HMI tags "Default tag table"
   "Any_Alm" : Bool = PLC Any_Alm AT %M6.7, 1 s
   "Reset_All" : Bool = PLC Reset_All AT %M4.1, 1 s
   "settings" : Int AT %DB1.DBW0
   "Any_Hand" : Bool = PLC Any_Hand AT %M5.0, 1 s
   "Logick_hand" : Bool = PLC Logic_DB.Hand AT %DB4.DBX526.7, 1 s
   "Valves_DB_V1_Status" : Int = PLC Valves_DB.V1.Status AT %DB3.DBW10, 1 s
   "Valves_DB_V2_Status" : Int = PLC Valves_DB.V2.Status AT %DB3.DBW134, 1 s
   "AOx_DB_SP_CF_Signal" : Int = PLC AOx_DB.T1_SP.Signal AT %DB8.DBW6, 1 s
   "AOx_DB_SP_CF_SP" : Real = PLC AOx_DB.T1_SP.SP AT %DB8.DBD0, 1 s
   "AOx_DB_SP_CF_CMD_Hand" : Bool = PLC AOx_DB.T1_SP.CMD.Hand AT %DB8.DBX8.0, 1 s
   "AOx_DB_SP_CF_SP_M" : Real = PLC AOx_DB.T1_SP.SP_M AT %DB8.DBD24, 1 s
   "Logic_DB_Start_weight" : Bool = PLC Logic_DB.Start_weight AT %DB4.DBX527.1, 1 s
   "Logic_DB_Alarm" : Word = PLC Logic_DB.Alarm AT %DB4.DBW528, 1 s
   "Motors_DB_T0_Alarm" : Word = PLC Motors_DB.T0.Alarm AT %DB2.DBW34, 1 s
   "Motors_DB_T1_Alarm" : Word = PLC Motors_DB.T1.Alarm AT %DB2.DBW78, 1 s
   "Motors_DB_T2_Alarm" : Word = PLC Motors_DB.T2.Alarm AT %DB2.DBW122, 1 s
   "Motors_DB_T3_Alarm" : Word = PLC Motors_DB.T3.Alarm AT %DB2.DBW166, 1 s
   "Motors_DB_T4_Alarm" : Word = PLC Motors_DB.T4.Alarm AT %DB2.DBW210, 1 s
   "Valves_DB_V1_Alarm" : Word = PLC Valves_DB.V1.Alarm AT %DB3.DBW70, 1 s
   "Valves_DB_V2_Alarm" : Word = PLC Valves_DB.V2.Alarm AT %DB3.DBW194, 1 s
   "Valves_DB_V3_Alarm" : Word = PLC Valves_DB.V3.Alarm AT %DB3.DBW318, 1 s
   "main_screens" : Int AT %DB1.DBW0
   "T4D4_DB_S1_SP" : Real = PLC T4D4_DB.S1.SP AT %DB10.DBD4, 1 s
   "Valves_DB_V1_Delay_On_SP" : Real = PLC Valves_DB.V1.Delay_On.SP AT %DB3.DBD30, 1 s
   "Valves_DB_V1_Delay_On_Now" : Real = PLC Valves_DB.V1.Delay_On.Now AT %DB3.DBD34, 1 s
   "Valves_DB_V1_Delay_Off_SP" : Real = PLC Valves_DB.V1.Delay_Off.SP AT %DB3.DBD48, 1 s
   "Valves_DB_V1_Delay_Off_Now" : Real = PLC Valves_DB.V1.Delay_Off.Now AT %DB3.DBD52, 1 s
   "Vis_reset_stat" : Bool AT %DB1.DBX0.0
   "T2D2_DB_Ready_T3D3" : Bool = PLC T2D2_DB.Ready_T3D3 AT %DB12.DBX0.1, 1 s
   "T3V3W3_DB_Skip_box" : Bool = PLC T3V3W3_DB.Skip_box AT %DB11.DBX8.6, 1 s
   "T3V3W3_DB_SetPoints_SP" : Real = PLC T3V3W3_DB.SetPoints.SP AT %DB11.DBD64, 1 s
   "T3V3W3_DB_LocalVar_SP_loaded" : Real = PLC T3V3W3_DB.LocalVar.SP_loaded AT %DB11.DBD92, 1 s
   "T3V3W3_DB_Reload" : Bool = PLC T3V3W3_DB.Reload AT %DB11.DBX6.4, 1 s
   "T3V3W3_DB_No_box" : Bool = PLC T3V3W3_DB.No_box AT %DB11.DBX8.7, 1 s
   "T3V3W3_DB_Timers_T_s7_SP" : Real = PLC T3V3W3_DB.Timers.T_s7.SP AT %DB11.DBD10, 1 s
   "T3V3W3_DB_Timers_T_s15_SP" : Real = PLC T3V3W3_DB.Timers.T_s15.SP AT %DB11.DBD28, 1 s
   "T3V3W3_DB_SetPoints_SP_ch_s" : Real = PLC T3V3W3_DB.SetPoints.SP_ch_s AT %DB11.DBD72, 1 s
   "T0T1_DB_SP_max" : Real = PLC T0T1_DB.SP_max AT %DB13.DBD8, 1 s
   "T0T1_DB_SP_min" : Real = PLC T0T1_DB.SP_min AT %DB13.DBD4, 1 s
   "T3V3W3_DB_SetPoints_SP_fly" : Real = PLC T3V3W3_DB.SetPoints.SP_fly AT %DB11.DBD68, 1 s
   "T3V3W3_DB_SetPoints_delta_add" : Real = PLC T3V3W3_DB.SetPoints.delta_add AT %DB11.DBD76, 1 s
   "T3V3W3_DB_SetPoints_delata_sub" : Real = PLC T3V3W3_DB.SetPoints.delata_sub AT %DB11.DBD80, 1 s
   "T3V3W3_DB_Reset_weight" : Bool = PLC T3V3W3_DB.Reset_weight AT %DB11.DBX8.4, 1 s
   "T3V3W3_DB_LocalVar_Sp_start" : Real = PLC T3V3W3_DB.LocalVar.Sp_start AT %DB11.DBD104, 1 s
   "Statistic_DB_move_stat_Instance_In_the_beggin" : Bool = PLC Statistic_DB.move_stat_Instance.In_the_beggin AT %DB19.DBX0.0, 1 s
   "Statistic_DB_move_stat_Instance_up" : Bool = PLC Statistic_DB.move_stat_Instance.up AT %DB19.DBX0.2, 1 s
   "T3V3W3_DB_Reset_statistic" : Bool = PLC T3V3W3_DB.Reset_statistic AT %DB11.DBX8.1, 1 s
   "Statistic_DB_move_stat_Instance_down" : Bool = PLC Statistic_DB.move_stat_Instance.down AT %DB19.DBX0.1, 1 s
   "Statistic_DB_move_stat_Instance_box_weight{1}" : Real = PLC Statistic_DB.move_stat_Instance.box_weight[1] AT %DB19.DBD2, 1 s
   "Statistic_DB_move_stat_Instance_box_weight{2}" : Real = PLC Statistic_DB.move_stat_Instance.box_weight[2] AT %DB19.DBD6, 1 s
   "Statistic_DB_move_stat_Instance_box_weight{3}" : Real = PLC Statistic_DB.move_stat_Instance.box_weight[3] AT %DB19.DBD10, 1 s
   "Statistic_DB_move_stat_Instance_box_weight{4}" : Real = PLC Statistic_DB.move_stat_Instance.box_weight[4] AT %DB19.DBD14, 1 s
   "Statistic_DB_move_stat_Instance_box_weight{5}" : Real = PLC Statistic_DB.move_stat_Instance.box_weight[5] AT %DB19.DBD18, 1 s
   "Statistic_DB_move_stat_Instance_box_weight{6}" : Real = PLC Statistic_DB.move_stat_Instance.box_weight[6] AT %DB19.DBD22, 1 s
   "Statistic_DB_move_stat_Instance_box_weight{7}" : Real = PLC Statistic_DB.move_stat_Instance.box_weight[7] AT %DB19.DBD26, 1 s
   "Statistic_DB_move_stat_Instance_box_weight{8}" : Real = PLC Statistic_DB.move_stat_Instance.box_weight[8] AT %DB19.DBD30, 1 s
   "Statistic_DB_move_stat_Instance_box_weight{9}" : Real = PLC Statistic_DB.move_stat_Instance.box_weight[9] AT %DB19.DBD34, 1 s
   "Statistic_DB_move_stat_Instance_box_weight{10}" : Real = PLC Statistic_DB.move_stat_Instance.box_weight[10] AT %DB19.DBD38, 1 s
   "Statistic_DB_move_stat_Instance_box_weight{11}" : Real = PLC Statistic_DB.move_stat_Instance.box_weight[11] AT %DB19.DBD42, 1 s
   "Statistic_DB_move_stat_Instance_box_weight{12}" : Real = PLC Statistic_DB.move_stat_Instance.box_weight[12] AT %DB19.DBD46, 1 s
   "Statistic_DB_move_stat_Instance_box_weight{13}" : Real = PLC Statistic_DB.move_stat_Instance.box_weight[13] AT %DB19.DBD50, 1 s
   "Statistic_DB_move_stat_Instance_box_weight{14}" : Real = PLC Statistic_DB.move_stat_Instance.box_weight[14] AT %DB19.DBD54, 1 s
   "Statistic_DB_move_stat_Instance_box_weight{15}" : Real = PLC Statistic_DB.move_stat_Instance.box_weight[15] AT %DB19.DBD58, 1 s
   "Statistic_DB_move_stat_Instance_box_weight{16}" : Real = PLC Statistic_DB.move_stat_Instance.box_weight[16] AT %DB19.DBD62, 1 s
   "Statistic_DB_move_stat_Instance_box_weight{17}" : Real = PLC Statistic_DB.move_stat_Instance.box_weight[17] AT %DB19.DBD66, 1 s
   "Statistic_DB_move_stat_Instance_box_weight{18}" : Real = PLC Statistic_DB.move_stat_Instance.box_weight[18] AT %DB19.DBD70, 1 s
   "Statistic_DB_move_stat_Instance_box_weight{19}" : Real = PLC Statistic_DB.move_stat_Instance.box_weight[19] AT %DB19.DBD74, 1 s
   "Statistic_DB_move_stat_Instance_box_weight{20}" : Real = PLC Statistic_DB.move_stat_Instance.box_weight[20] AT %DB19.DBD78, 1 s
   "Statistic_DB_move_stat_Instance_box_weight{21}" : Real = PLC Statistic_DB.move_stat_Instance.box_weight[21] AT %DB19.DBD82, 1 s
   "Statistic_DB_move_stat_Instance_box_weight{22}" : Real = PLC Statistic_DB.move_stat_Instance.box_weight[22] AT %DB19.DBD86, 1 s
   "Statistic_DB_move_stat_Instance_box_weight{23}" : Real = PLC Statistic_DB.move_stat_Instance.box_weight[23] AT %DB19.DBD90, 1 s
   "Statistic_DB_move_stat_Instance_box_weight{24}" : Real = PLC Statistic_DB.move_stat_Instance.box_weight[24] AT %DB19.DBD94, 1 s
   "Statistic_DB_move_stat_Instance_box_weight{25}" : Real = PLC Statistic_DB.move_stat_Instance.box_weight[25] AT %DB19.DBD98, 1 s
   "T3V3W3_DB_Statistic_Count" : Int = PLC T3V3W3_DB.Statistic.Count AT %DB11.DBW378, 1 s
   "T3V3W3_DB_Statistic_Mid_weight" : Real = PLC T3V3W3_DB.Statistic.Mid_weight AT %DB11.DBD384, 1 s
   "T3V3W3_DB_Statistic_Weight" : Real = PLC T3V3W3_DB.Statistic.Weight AT %DB11.DBD380, 1 s
   "T3V3W3_DB_Statistic_Count_old" : Int = PLC T3V3W3_DB.Statistic.Count_old AT %DB11.DBW388, 1 s
   "T3V3W3_DB_Statistic_Mid_weight_old" : Real = PLC T3V3W3_DB.Statistic.Mid_weight_old AT %DB11.DBD394, 1 s
   "T3V3W3_DB_Statistic_Weight_old" : Real = PLC T3V3W3_DB.Statistic.Weight_old AT %DB11.DBD390, 1 s
   "T3V3W3_DB_Alarm" : Word = PLC T3V3W3_DB.Alarm AT %DB11.DBW404, 1 s
   "T3V3W3_DB_LocalVar_name_part" : String[254] = PLC T3V3W3_DB.LocalVar.name_part AT %DB11.DBX118.0, 1 s
   "Logic_DB_Clear_mem" : Bool = PLC Logic_DB.Clear_mem AT %DB4.DBX2.0, 1 s
   "T3V3W3_DB_part_names{0}" : String[254] = PLC T3V3W3_DB.part_names[0] AT %DB11.DBX422.0, 1 s
   "T3V3W3_DB_part_names{1}" : String[254] = PLC T3V3W3_DB.part_names[1] AT %DB11.DBX678.0, 1 s
   "T3V3W3_DB_part_names{2}" : String[254] = PLC T3V3W3_DB.part_names[2] AT %DB11.DBX934.0, 1 s
   "T3V3W3_DB_part_names{3}" : String[254] = PLC T3V3W3_DB.part_names[3] AT %DB11.DBX1190.0, 1 s
   "T3V3W3_DB_part_names{4}" : String[254] = PLC T3V3W3_DB.part_names[4] AT %DB11.DBX1446.0, 1 s
   "T3V3W3_DB_part_names{5}" : String[254] = PLC T3V3W3_DB.part_names[5] AT %DB11.DBX1702.0, 1 s
   "T3V3W3_DB_part_names{6}" : String[254] = PLC T3V3W3_DB.part_names[6] AT %DB11.DBX1958.0, 1 s
   "T3V3W3_DB_part_names{7}" : String[254] = PLC T3V3W3_DB.part_names[7] AT %DB11.DBX2214.0, 1 s
   "T3V3W3_DB_part_names{8}" : String[254] = PLC T3V3W3_DB.part_names[8] AT %DB11.DBX2470.0, 1 s
   "T3V3W3_DB_part_names{9}" : String[254] = PLC T3V3W3_DB.part_names[9] AT %DB11.DBX2726.0, 1 s
   "T3V3W3_DB_part_names{10}" : String[254] = PLC T3V3W3_DB.part_names[10] AT %DB11.DBX2982.0, 1 s
   "T3V3W3_DB_part_names{11}" : String[254] = PLC T3V3W3_DB.part_names[11] AT %DB11.DBX3238.0, 1 s
   "T3V3W3_DB_part_names{12}" : String[254] = PLC T3V3W3_DB.part_names[12] AT %DB11.DBX3494.0, 1 s
   "T3V3W3_DB_part_names{13}" : String[254] = PLC T3V3W3_DB.part_names[13] AT %DB11.DBX3750.0, 1 s
   "T3V3W3_DB_part_names{14}" : String[254] = PLC T3V3W3_DB.part_names[14] AT %DB11.DBX4006.0, 1 s
   "T3V3W3_DB_part_names{15}" : String[254] = PLC T3V3W3_DB.part_names[15] AT %DB11.DBX4262.0, 1 s
   "T3V3W3_DB_part_names{16}" : String[254] = PLC T3V3W3_DB.part_names[16] AT %DB11.DBX4518.0, 1 s
   "T3V3W3_DB_part_names{17}" : String[254] = PLC T3V3W3_DB.part_names[17] AT %DB11.DBX4774.0, 1 s
   "T3V3W3_DB_part_names{18}" : String[254] = PLC T3V3W3_DB.part_names[18] AT %DB11.DBX5030.0, 1 s
   "T3V3W3_DB_part_names{19}" : String[254] = PLC T3V3W3_DB.part_names[19] AT %DB11.DBX5286.0, 1 s
   "del_stat_mem_DB_del" : Bool = PLC del_stat_mem_DB.del AT %DB14.DBX0.2, 1 s
   "del_stat_mem_DB_number" : Int = PLC del_stat_mem_DB.number AT %DB14.DBW4, 1 s
   "del_stat_mem_DB_Alarm" : Word = PLC del_stat_mem_DB.Alarm AT %DB14.DBW550, 1 s
   "stat_view" : Int AT %DB1.DBW0
   "T3V3W3_DB_Timers_T_St_Start" : Bool = PLC T3V3W3_DB.Timers.T_St.Start AT %DB11.DBX62.1, 1 s

HMI tags "motors"
   "T0_CMD_Hand" : Bool = PLC Motors_DB.T0.CMD.Hand AT %DB2.DBX6.0, 1 s
   "T0_CMD_Force" : Bool = PLC Motors_DB.T0.CMD.Force AT %DB2.DBX6.3, 1 s
   "T0_Res_h" : DInt = PLC Motors_DB.T0.Res_h AT %DB2.DBD36, 1 s
   "T0_Wait_Off_SP" : Int = PLC Motors_DB.T0.Wait_Off.SP AT %DB2.DBW24, 1 s
   "T0_Wait_Off_Now" : Int = PLC Motors_DB.T0.Wait_Off.Now AT %DB2.DBW26, 1 s
   "T0_Wait_On_SP" : Int = PLC Motors_DB.T0.Wait_On.SP AT %DB2.DBW18, 1 s
   "T0_Wait_On_Now" : Int = PLC Motors_DB.T0.Wait_On.Now AT %DB2.DBW20, 1 s
   "T0_FB_Termo" : Bool = PLC Motors_DB.T0.FB_Termo AT %DB2.DBX0.3, 1 s
   "T0_Use_Termo" : Bool = PLC Motors_DB.T0.Use.Termo AT %DB2.DBX12.4, 1 s
   "T0_Use_Serivce" : Bool = PLC Motors_DB.T0.Use.Serivce AT %DB2.DBX12.3, 1 s
   "T0_Use_KM" : Bool = PLC Motors_DB.T0.Use.KM AT %DB2.DBX12.2, 1 s
   "T0_Use_QF" : Bool = PLC Motors_DB.T0.Use.QF AT %DB2.DBX12.1, 1 s
   "T1_CMD_Hand" : Bool = PLC Motors_DB.T1.CMD.Hand AT %DB2.DBX50.0, 1 s
   "T1_CMD_Force" : Bool = PLC Motors_DB.T1.CMD.Force AT %DB2.DBX50.3, 1 s
   "T1_Res_h" : DInt = PLC Motors_DB.T1.Res_h AT %DB2.DBD80, 1 s
   "T1_Wait_Off_SP" : Int = PLC Motors_DB.T1.Wait_Off.SP AT %DB2.DBW68, 1 s
   "T1_Wait_Off_Now" : Int = PLC Motors_DB.T1.Wait_Off.Now AT %DB2.DBW70, 1 s
   "T1_Wait_On_SP" : Int = PLC Motors_DB.T1.Wait_On.SP AT %DB2.DBW62, 1 s
   "T1_Wait_On_Now" : Int = PLC Motors_DB.T1.Wait_On.Now AT %DB2.DBW64, 1 s
   "T1_FB_Termo" : Bool = PLC Motors_DB.T1.FB_Termo AT %DB2.DBX44.3, 1 s
   "T1_Use_Termo" : Bool = PLC Motors_DB.T1.Use.Termo AT %DB2.DBX56.4, 1 s
   "T1_Use_Serivce" : Bool = PLC Motors_DB.T1.Use.Serivce AT %DB2.DBX56.3, 1 s
   "T1_Use_KM" : Bool = PLC Motors_DB.T1.Use.KM AT %DB2.DBX56.2, 1 s
   "T1_Use_QF" : Bool = PLC Motors_DB.T1.Use.QF AT %DB2.DBX56.1, 1 s
   "T3_CMD_Hand" : Bool = PLC Motors_DB.T3.CMD.Hand AT %DB2.DBX138.0, 1 s
   "T3_CMD_Force" : Bool = PLC Motors_DB.T3.CMD.Force AT %DB2.DBX138.3, 1 s
   "T3_Res_h" : DInt = PLC Motors_DB.T3.Res_h AT %DB2.DBD168, 1 s
   "T3_Wait_Off_SP" : Int = PLC Motors_DB.T3.Wait_Off.SP AT %DB2.DBW156, 1 s
   "T3_Wait_Off_Now" : Int = PLC Motors_DB.T3.Wait_Off.Now AT %DB2.DBW158, 1 s
   "T3_FB_Termo" : Bool = PLC Motors_DB.T3.FB_Termo AT %DB2.DBX132.3, 1 s
   "T3_Use_Termo" : Bool = PLC Motors_DB.T3.Use.Termo AT %DB2.DBX144.4, 1 s
   "T3_Use_Serivce" : Bool = PLC Motors_DB.T3.Use.Serivce AT %DB2.DBX144.3, 1 s
   "T3_Use_KM" : Bool = PLC Motors_DB.T3.Use.KM AT %DB2.DBX144.2, 1 s
   "T3_Use_QF" : Bool = PLC Motors_DB.T3.Use.QF AT %DB2.DBX144.1, 1 s
   "T2_CMD_Hand" : Bool = PLC Motors_DB.T2.CMD.Hand AT %DB2.DBX94.0, 1 s
   "T2_CMD_Force" : Bool = PLC Motors_DB.T2.CMD.Force AT %DB2.DBX94.3, 1 s
   "T2_Res_h" : DInt = PLC Motors_DB.T2.Res_h AT %DB2.DBD124, 1 s
   "T2_Wait_Off_Now" : Int = PLC Motors_DB.T2.Wait_Off.Now AT %DB2.DBW114, 1 s
   "T2_Wait_Off_SP" : Int = PLC Motors_DB.T2.Wait_Off.SP AT %DB2.DBW112, 1 s
   "T2_Wait_On_SP" : Int = PLC Motors_DB.T2.Wait_On.SP AT %DB2.DBW106, 1 s
   "T2_Wait_On_Now" : Int = PLC Motors_DB.T2.Wait_On.Now AT %DB2.DBW108, 1 s
   "T2_FB_Termo" : Bool = PLC Motors_DB.T2.FB_Termo AT %DB2.DBX88.3, 1 s
   "T2_Use_Termo" : Bool = PLC Motors_DB.T2.Use.Termo AT %DB2.DBX100.4, 1 s
   "T2_Use_Serivce" : Bool = PLC Motors_DB.T2.Use.Serivce AT %DB2.DBX100.3, 1 s
   "T2_Use_KM" : Bool = PLC Motors_DB.T2.Use.KM AT %DB2.DBX100.2, 1 s
   "T2_Use_QF" : Bool = PLC Motors_DB.T2.Use.QF AT %DB2.DBX100.1, 1 s
   "T3_Wait_On_SP" : Int = PLC Motors_DB.T3.Wait_On.SP AT %DB2.DBW150, 1 s
   "T3_Wait_On_Now" : Int = PLC Motors_DB.T3.Wait_On.Now AT %DB2.DBW152, 1 s
   "T3_FB_QF" : Bool = PLC Motors_DB.T3.FB_QF AT %DB2.DBX132.0, 1 s
   "T3_FB_KM" : Bool = PLC Motors_DB.T3.FB_KM AT %DB2.DBX132.1, 1 s
   "T3_CMD_Service" : Bool = PLC Motors_DB.T3.CMD.Service AT %DB2.DBX138.6, 1 s
   "T3_CMD_Sim" : Bool = PLC Motors_DB.T3.CMD.Sim AT %DB2.DBX139.2, 1 s
   "T3_Status" : Int = PLC Motors_DB.T3.Status AT %DB2.DBW142, 1 s
   "T3_CMD_Start_M" : Bool = PLC Motors_DB.T3.CMD.Start_M AT %DB2.DBX138.2, 1 s
   "T1_FB_QF" : Bool = PLC Motors_DB.T1.FB_QF AT %DB2.DBX44.0, 1 s
   "T1_FB_KM" : Bool = PLC Motors_DB.T1.FB_KM AT %DB2.DBX44.1, 1 s
   "T1_Status" : Int = PLC Motors_DB.T1.Status AT %DB2.DBW54, 1 s
   "T1_CMD_Sim" : Bool = PLC Motors_DB.T1.CMD.Sim AT %DB2.DBX51.2, 1 s
   "T1_CMD_Start_M" : Bool = PLC Motors_DB.T1.CMD.Start_M AT %DB2.DBX50.2, 1 s
   "T0_FB_QF" : Bool = PLC Motors_DB.T0.FB_QF AT %DB2.DBX0.0, 1 s
   "T0_FB_KM" : Bool = PLC Motors_DB.T0.FB_KM AT %DB2.DBX0.1, 1 s
   "T0_CMD_Sim" : Bool = PLC Motors_DB.T0.CMD.Sim AT %DB2.DBX7.2, 1 s
   "T0_CMD_Start_M" : Bool = PLC Motors_DB.T0.CMD.Start_M AT %DB2.DBX6.2, 1 s
   "T0_Status" : Int = PLC Motors_DB.T0.Status AT %DB2.DBW10, 1 s
   "T2_FB_QF" : Bool = PLC Motors_DB.T2.FB_QF AT %DB2.DBX88.0, 1 s
   "T2_FB_KM" : Bool = PLC Motors_DB.T2.FB_KM AT %DB2.DBX88.1, 1 s
   "T2_CMD_Start_M" : Bool = PLC Motors_DB.T2.CMD.Start_M AT %DB2.DBX94.2, 1 s
   "T2_CMD_Sim" : Bool = PLC Motors_DB.T2.CMD.Sim AT %DB2.DBX95.2, 1 s
   "T2_Status" : Int = PLC Motors_DB.T2.Status AT %DB2.DBW98, 1 s
   "T0_CMD_Service" : Bool = PLC Motors_DB.T0.CMD.Service AT %DB2.DBX6.6, 1 s
   "T1_CMD_Service" : Bool = PLC Motors_DB.T1.CMD.Service AT %DB2.DBX50.6, 1 s
   "T2_CMD_Service" : Bool = PLC Motors_DB.T2.CMD.Service AT %DB2.DBX94.6, 1 s
   "T4_FB_QF" : Bool = PLC Motors_DB.T4.FB_QF AT %DB2.DBX176.0, 1 s
   "T4_FB_KM" : Bool = PLC Motors_DB.T4.FB_KM AT %DB2.DBX176.1, 1 s
   "T4_FB_Service" : Bool = PLC Motors_DB.T4.FB_Service AT %DB2.DBX176.2, 1 s
   "T4_FB_Termo" : Bool = PLC Motors_DB.T4.FB_Termo AT %DB2.DBX176.3, 1 s
   "T4_CMD_Hand" : Bool = PLC Motors_DB.T4.CMD.Hand AT %DB2.DBX182.0, 1 s
   "T4_CMD_Start_A" : Bool = PLC Motors_DB.T4.CMD.Start_A AT %DB2.DBX182.1, 1 s
   "T4_CMD_Start_M" : Bool = PLC Motors_DB.T4.CMD.Start_M AT %DB2.DBX182.2, 1 s
   "T4_CMD_Force" : Bool = PLC Motors_DB.T4.CMD.Force AT %DB2.DBX182.3, 1 s
   "T4_CMD_Local" : Bool = PLC Motors_DB.T4.CMD.Local AT %DB2.DBX182.5, 1 s
   "T4_CMD_Safety" : Bool = PLC Motors_DB.T4.CMD.Safety AT %DB2.DBX182.7, 1 s
   "T4_CMD_Service" : Bool = PLC Motors_DB.T4.CMD.Service AT %DB2.DBX182.6, 1 s
   "T4_CMD_Sim" : Bool = PLC Motors_DB.T4.CMD.Sim AT %DB2.DBX183.2, 1 s
   "T4_Status" : Int = PLC Motors_DB.T4.Status AT %DB2.DBW186, 1 s
   "T4_Use_QF" : Bool = PLC Motors_DB.T4.Use.QF AT %DB2.DBX188.1, 1 s
   "T4_Use_KM" : Bool = PLC Motors_DB.T4.Use.KM AT %DB2.DBX188.2, 1 s
   "T4_Use_Serivce" : Bool = PLC Motors_DB.T4.Use.Serivce AT %DB2.DBX188.3, 1 s
   "T4_Use_Termo" : Bool = PLC Motors_DB.T4.Use.Termo AT %DB2.DBX188.4, 1 s
   "T4_FB_QF(1)" : Bool = PLC Motors_DB.T4.FB.QF AT %DB2.DBX190.1, 1 s
   "T4_FB_KM(1)" : Bool = PLC Motors_DB.T4.FB.KM AT %DB2.DBX190.2, 1 s
   "T4_FB_Serivce" : Bool = PLC Motors_DB.T4.FB.Serivce AT %DB2.DBX190.3, 1 s
   "T4_FB_Termo(1)" : Bool = PLC Motors_DB.T4.FB.Termo AT %DB2.DBX190.4, 1 s
   "T4_Wait_On_SP" : Int = PLC Motors_DB.T4.Wait_On.SP AT %DB2.DBW194, 1 s
   "T4_Wait_On_Now" : Int = PLC Motors_DB.T4.Wait_On.Now AT %DB2.DBW196, 1 s
   "T4_Wait_Off_SP" : Int = PLC Motors_DB.T4.Wait_Off.SP AT %DB2.DBW200, 1 s
   "T4_Wait_Off_Now" : Int = PLC Motors_DB.T4.Wait_Off.Now AT %DB2.DBW202, 1 s
   "T4_Res_h" : DInt = PLC Motors_DB.T4.Res_h AT %DB2.DBD212, 1 s

HMI tags "Valves"
   "V1_Status" : Int = PLC Valves_DB.V1.Status AT %DB3.DBW10, 1 s
   "V1_CMD_Force" : Bool = PLC Valves_DB.V1.CMD.Force AT %DB3.DBX6.3, 1 s
   "V1_Wait_On_SP" : Int = PLC Valves_DB.V1.Wait_On.SP AT %DB3.DBW18, 1 s
   "V1_Wait_On_Now" : Int = PLC Valves_DB.V1.Wait_On.Now AT %DB3.DBW20, 1 s
   "V1_CMD_Start_A" : Bool = PLC Valves_DB.V1.CMD.Start_A AT %DB3.DBX6.1, 1 s
   "V1_CMD_Start_M" : Bool = PLC Valves_DB.V1.CMD.Start_M AT %DB3.DBX6.2, 1 s
   "V1_CMD_Hand" : Bool = PLC Valves_DB.V1.CMD.Hand AT %DB3.DBX6.0, 1 s
   "V1_CMD_Service" : Bool = PLC Valves_DB.V1.CMD.Service AT %DB3.DBX6.6, 1 s
   "V1_CMD_Local" : Bool = PLC Valves_DB.V1.CMD.Local AT %DB3.DBX6.5, 1 s
   "V1_Use_QF" : Bool = PLC Valves_DB.V1.Use.QF AT %DB3.DBX12.1, 1 s
   "V1_Use_Serivce" : Bool = PLC Valves_DB.V1.Use.Serivce AT %DB3.DBX12.4, 1 s
   "V1_Use_Open" : Bool = PLC Valves_DB.V1.Use.Open AT %DB3.DBX12.5, 1 s
   "V1_Use_Close" : Bool = PLC Valves_DB.V1.Use.Close AT %DB3.DBX12.6, 1 s
   "V1_FB_QF" : Bool = PLC Valves_DB.V1.FB_QF AT %DB3.DBX0.0, 1 s
   "V1_FB_Open" : Bool = PLC Valves_DB.V1.FB_Open AT %DB3.DBX0.4, 1 s
   "V1_FB_Close" : Bool = PLC Valves_DB.V1.FB_Close AT %DB3.DBX0.5, 1 s
   "V1_FB_Service" : Bool = PLC Valves_DB.V1.FB_Service AT %DB3.DBX0.3, 1 s
   "V1_CMD_Sim" : Bool = PLC Valves_DB.V1.CMD.Sim AT %DB3.DBX7.2, 1 s
   "V1_Res_h" : DInt = PLC Valves_DB.V1.Res_h AT %DB3.DBD72, 1 s
   "V2_FB_QF" : Bool = PLC Valves_DB.V2.FB_QF AT %DB3.DBX124.0, 1 s
   "V2_FB_Service" : Bool = PLC Valves_DB.V2.FB_Service AT %DB3.DBX124.3, 1 s
   "V2_FB_Open" : Bool = PLC Valves_DB.V2.FB_Open AT %DB3.DBX124.4, 1 s
   "V2_FB_Close" : Bool = PLC Valves_DB.V2.FB_Close AT %DB3.DBX124.5, 1 s
   "V2_CMD_Hand" : Bool = PLC Valves_DB.V2.CMD.Hand AT %DB3.DBX130.0, 1 s
   "V2_CMD_Start_M" : Bool = PLC Valves_DB.V2.CMD.Start_M AT %DB3.DBX130.2, 1 s
   "V2_CMD_Force" : Bool = PLC Valves_DB.V2.CMD.Force AT %DB3.DBX130.3, 1 s
   "V2_CMD_Service" : Bool = PLC Valves_DB.V2.CMD.Service AT %DB3.DBX130.6, 1 s
   "V2_CMD_Sim" : Bool = PLC Valves_DB.V2.CMD.Sim AT %DB3.DBX131.2, 1 s
   "V2_Use_QF" : Bool = PLC Valves_DB.V2.Use.QF AT %DB3.DBX136.1, 1 s
   "V2_Use_Serivce" : Bool = PLC Valves_DB.V2.Use.Serivce AT %DB3.DBX136.4, 1 s
   "V2_Use_Open" : Bool = PLC Valves_DB.V2.Use.Open AT %DB3.DBX136.5, 1 s
   "V2_Use_Close" : Bool = PLC Valves_DB.V2.Use.Close AT %DB3.DBX136.6, 1 s
   "V2_FB_QF(1)" : Bool = PLC Valves_DB.V2.FB.QF AT %DB3.DBX138.1, 1 s
   "V2_FB_Open(1)" : Bool = PLC Valves_DB.V2.FB.Open AT %DB3.DBX138.5, 1 s
   "V2_FB_Close(1)" : Bool = PLC Valves_DB.V2.FB.Close AT %DB3.DBX138.6, 1 s
   "V2_FB_Serivce" : Bool = PLC Valves_DB.V2.FB.Serivce AT %DB3.DBX138.4, 1 s
   "V2_Wait_On_SP" : Int = PLC Valves_DB.V2.Wait_On.SP AT %DB3.DBW142, 1 s
   "V2_Wait_On_Now" : Int = PLC Valves_DB.V2.Wait_On.Now AT %DB3.DBW144, 1 s
   "V2_Wait_Off_SP" : Int = PLC Valves_DB.V2.Wait_Off.SP AT %DB3.DBW148, 1 s
   "V2_Wait_Off_Now" : Int = PLC Valves_DB.V2.Wait_Off.Now AT %DB3.DBW150, 1 s
   "V2_Res_h" : DInt = PLC Valves_DB.V2.Res_h AT %DB3.DBD196, 1 s
   "V1_Wait_Off_SP" : Int = PLC Valves_DB.V1.Wait_Off.SP AT %DB3.DBW24, 1 s
   "V1_Wait_Off_Now" : Int = PLC Valves_DB.V1.Wait_Off.Now AT %DB3.DBW26, 1 s
   "V3_FB_QF" : Bool = PLC Valves_DB.V3.FB_QF AT %DB3.DBX248.0, 1 s
   "V3_FB_Open" : Bool = PLC Valves_DB.V3.FB_Open AT %DB3.DBX248.4, 1 s
   "V3_FB_Close" : Bool = PLC Valves_DB.V3.FB_Close AT %DB3.DBX248.5, 1 s
   "V3_FB_Service" : Bool = PLC Valves_DB.V3.FB_Service AT %DB3.DBX248.3, 1 s
   "V3_CMD_Start_A" : Bool = PLC Valves_DB.V3.CMD.Start_A AT %DB3.DBX254.1, 1 s
   "V3_CMD_Start_M" : Bool = PLC Valves_DB.V3.CMD.Start_M AT %DB3.DBX254.2, 1 s
   "V3_CMD_Hand" : Bool = PLC Valves_DB.V3.CMD.Hand AT %DB3.DBX254.0, 1 s
   "V3_CMD_Force" : Bool = PLC Valves_DB.V3.CMD.Force AT %DB3.DBX254.3, 1 s
   "V3_CMD_Sim" : Bool = PLC Valves_DB.V3.CMD.Sim AT %DB3.DBX255.2, 1 s
   "V3_Status" : Int = PLC Valves_DB.V3.Status AT %DB3.DBW258, 1 s
   "V3_FB_QF(1)" : Bool = PLC Valves_DB.V3.FB.QF AT %DB3.DBX262.1, 1 s
   "V3_FB_Serivce" : Bool = PLC Valves_DB.V3.FB.Serivce AT %DB3.DBX262.4, 1 s
   "V3_FB_Open(1)" : Bool = PLC Valves_DB.V3.FB.Open AT %DB3.DBX262.5, 1 s
   "V3_FB_Close(1)" : Bool = PLC Valves_DB.V3.FB.Close AT %DB3.DBX262.6, 1 s
   "V3_Wait_On_SP" : Int = PLC Valves_DB.V3.Wait_On.SP AT %DB3.DBW266, 1 s
   "V3_Wait_On_Now" : Int = PLC Valves_DB.V3.Wait_On.Now AT %DB3.DBW268, 1 s
   "V3_Wait_Off_SP" : Int = PLC Valves_DB.V3.Wait_Off.SP AT %DB3.DBW272, 1 s
   "V3_Wait_Off_Now" : Int = PLC Valves_DB.V3.Wait_Off.Now AT %DB3.DBW274, 1 s
   "V3_Res_h" : DInt = PLC Valves_DB.V3.Res_h AT %DB3.DBD320, 1 s
   "V3_CMD_Service" : Bool = PLC Valves_DB.V3.CMD.Service AT %DB3.DBX254.6, 1 s
   "V3_Use_QF" : Bool = PLC Valves_DB.V3.Use.QF AT %DB3.DBX260.1, 1 s
   "V3_Use_Open" : Bool = PLC Valves_DB.V3.Use.Open AT %DB3.DBX260.5, 1 s
   "V3_Use_Close" : Bool = PLC Valves_DB.V3.Use.Close AT %DB3.DBX260.6, 1 s
   "V3_Use_Serivce" : Bool = PLC Valves_DB.V3.Use.Serivce AT %DB3.DBX260.4, 1 s
   "Valves_DB_V2_Delay_On_SP" : Real = PLC Valves_DB.V2.Delay_On.SP AT %DB3.DBD154, 1 s
   "Valves_DB_V2_Delay_On_Now" : Real = PLC Valves_DB.V2.Delay_On.Now AT %DB3.DBD158, 1 s
   "Valves_DB_V2_Delay_Off_SP" : Real = PLC Valves_DB.V2.Delay_Off.SP AT %DB3.DBD172, 1 s
   "Valves_DB_V2_Delay_Off_Now" : Real = PLC Valves_DB.V2.Delay_Off.Now AT %DB3.DBD176, 1 s
   "Valves_DB_V3_Delay_On_SP" : Real = PLC Valves_DB.V3.Delay_On.SP AT %DB3.DBD278, 1 s
   "Valves_DB_V3_Delay_On_Now" : Real = PLC Valves_DB.V3.Delay_On.Now AT %DB3.DBD282, 1 s
   "Valves_DB_V3_Delay_Off_SP" : Real = PLC Valves_DB.V3.Delay_Off.SP AT %DB3.DBD296, 1 s
   "Valves_DB_V3_Delay_Off_Now" : Real = PLC Valves_DB.V3.Delay_Off.Now AT %DB3.DBD300, 1 s

HMI tags "DIx"
   "Voltage_CPU_Ok_Input" : Bool = PLC DIx_DB.Voltage_CPU_Ok.Input AT %DB9.DBX0.0, 1 s
   "Voltage_CPU_Ok_Signal" : Bool = PLC DIx_DB.Voltage_CPU_Ok.Signal AT %DB9.DBX2.0, 1 s
   "Voltage_CPU_Ok_Start_M" : Bool = PLC DIx_DB.Voltage_CPU_Ok.Start_M AT %DB9.DBX4.1, 1 s
   "Voltage_CPU_Ok_Hand" : Bool = PLC DIx_DB.Voltage_CPU_Ok.Hand AT %DB9.DBX4.0, 1 s
   "Voltage_CPU_Ok_Inverse" : Bool = PLC DIx_DB.Voltage_CPU_Ok.Inverse AT %DB9.DBX4.3, 1 s
   "Voltage_CPU_Ok_Filter_On_SP" : Int = PLC DIx_DB.Voltage_CPU_Ok.Filter_On.SP AT %DB9.DBW6, 1 s
   "Voltage_CPU_Ok_Filter_Off_SP" : Int = PLC DIx_DB.Voltage_CPU_Ok.Filter_Off.SP AT %DB9.DBW12, 1 s
   "Voltage_DI_Ok_Input" : Bool = PLC DIx_DB.Voltage_DI_Ok.Input AT %DB9.DBX20.0, 1 s
   "Voltage_DI_Ok_Signal" : Bool = PLC DIx_DB.Voltage_DI_Ok.Signal AT %DB9.DBX22.0, 1 s
   "Voltage_DI_Ok_Hand" : Bool = PLC DIx_DB.Voltage_DI_Ok.Hand AT %DB9.DBX24.0, 1 s
   "Voltage_DI_Ok_Start_M" : Bool = PLC DIx_DB.Voltage_DI_Ok.Start_M AT %DB9.DBX24.1, 1 s
   "Voltage_DI_Ok_Inverse" : Bool = PLC DIx_DB.Voltage_DI_Ok.Inverse AT %DB9.DBX24.3, 1 s
   "Voltage_DI_Ok_Filter_On_SP" : Int = PLC DIx_DB.Voltage_DI_Ok.Filter_On.SP AT %DB9.DBW26, 1 s
   "Voltage_DI_Ok_Filter_Off_SP" : Int = PLC DIx_DB.Voltage_DI_Ok.Filter_Off.SP AT %DB9.DBW32, 1 s
   "Voltage_DO_Ok_Input" : Bool = PLC DIx_DB.Voltage_DO_Ok.Input AT %DB9.DBX40.0, 1 s
   "Voltage_DO_Ok_Signal" : Bool = PLC DIx_DB.Voltage_DO_Ok.Signal AT %DB9.DBX42.0, 1 s
   "Voltage_DO_Ok_Hand" : Bool = PLC DIx_DB.Voltage_DO_Ok.Hand AT %DB9.DBX44.0, 1 s
   "Voltage_DO_Ok_Start_M" : Bool = PLC DIx_DB.Voltage_DO_Ok.Start_M AT %DB9.DBX44.1, 1 s
   "Voltage_DO_Ok_Inverse" : Bool = PLC DIx_DB.Voltage_DO_Ok.Inverse AT %DB9.DBX44.3, 1 s
   "Voltage_DO_Ok_Filter_On_SP" : Int = PLC DIx_DB.Voltage_DO_Ok.Filter_On.SP AT %DB9.DBW46, 1 s
   "Voltage_DO_Ok_Filter_Off_SP" : Int = PLC DIx_DB.Voltage_DO_Ok.Filter_Off.SP AT %DB9.DBW52, 1 s
   "Voltage_24V_Ok_Input" : Bool = PLC DIx_DB.Voltage_24V_Ok.Input AT %DB9.DBX60.0, 1 s
   "Voltage_24V_Ok_Signal" : Bool = PLC DIx_DB.Voltage_24V_Ok.Signal AT %DB9.DBX62.0, 1 s
   "Voltage_24V_Ok_Hand" : Bool = PLC DIx_DB.Voltage_24V_Ok.Hand AT %DB9.DBX64.0, 1 s
   "Voltage_24V_Ok_Start_M" : Bool = PLC DIx_DB.Voltage_24V_Ok.Start_M AT %DB9.DBX64.1, 1 s
   "Voltage_24V_Ok_Inverse" : Bool = PLC DIx_DB.Voltage_24V_Ok.Inverse AT %DB9.DBX64.3, 1 s
   "Voltage_24V_Ok_Filter_On_SP" : Int = PLC DIx_DB.Voltage_24V_Ok.Filter_On.SP AT %DB9.DBW66, 1 s
   "Voltage_24V_Ok_Filter_Off_SP" : Int = PLC DIx_DB.Voltage_24V_Ok.Filter_Off.SP AT %DB9.DBW72, 1 s
   "Safety_Ok_Input" : Bool = PLC DIx_DB.Safety_Ok.Input AT %DB9.DBX80.0, 1 s
   "Safety_Ok_Signal" : Bool = PLC DIx_DB.Safety_Ok.Signal AT %DB9.DBX82.0, 1 s
   "Safety_Ok_Hand" : Bool = PLC WP231PR_DB.DR06.DELAY_EMPTY AT %DB9.DBX84.0, 1 s
   "Safety_Ok_Start_M" : Bool = PLC DIx_DB.Safety_Ok.Start_M AT %DB9.DBX84.1, 1 s
   "Safety_Ok_Inverse" : Bool = PLC DIx_DB.Safety_Ok.Inverse AT %DB9.DBX84.3, 1 s
   "Safety_Ok_Filter_On_SP" : Int = PLC DIx_DB.Safety_Ok.Filter_On.SP AT %DB9.DBW86, 1 s
   "Safety_Ok_Filter_Off_SP" : Int = PLC DIx_DB.Safety_Ok.Filter_Off.SP AT %DB9.DBW92, 1 s
   "Cold_tunnel_QF_Input" : Bool = PLC DIx_DB.Cold_tunnel_QF.Input AT %DB9.DBX100.0, 1 s
   "Cold_tunnel_QF_Signal" : Bool = PLC DIx_DB.Cold_tunnel_QF.Signal AT %DB9.DBX102.0, 1 s
   "Cold_tunnel_QF_Hand" : Bool = PLC DIx_DB.Cold_tunnel_QF.Hand AT %DB9.DBX104.0, 1 s
   "Cold_tunnel_QF_Start_M" : Bool = PLC DIx_DB.Cold_tunnel_QF.Start_M AT %DB9.DBX104.1, 1 s
   "Cold_tunnel_QF_Inverse" : Bool = PLC DIx_DB.Cold_tunnel_QF.Inverse AT %DB9.DBX104.3, 1 s
   "Cold_tunnel_QF_Filter_On_SP" : Int = PLC DIx_DB.Cold_tunnel_QF.Filter_On.SP AT %DB9.DBW106, 1 s
   "Cold_tunnel_QF_Filter_Off_SP" : Int = PLC DIx_DB.Cold_tunnel_QF.Filter_Off.SP AT %DB9.DBW112, 1 s
   "T1_QF_Input" : Bool = PLC DIx_DB.T1_QF.Input AT %DB9.DBX120.0, 1 s
   "T1_QF_Signal" : Bool = PLC DIx_DB.T1_QF.Signal AT %DB9.DBX122.0, 1 s
   "T1_QF_Hand" : Bool = PLC DIx_DB.T1_QF.Hand AT %DB9.DBX124.0, 1 s
   "T1_QF_Start_M" : Bool = PLC DIx_DB.T1_QF.Start_M AT %DB9.DBX124.1, 1 s
   "T1_QF_Inverse" : Bool = PLC DIx_DB.T1_QF.Inverse AT %DB9.DBX124.3, 1 s
   "T1_QF_Filter_On_SP" : Int = PLC DIx_DB.T1_QF.Filter_On.SP AT %DB9.DBW126, 1 s
   "T1_QF_Filter_Off_SP" : Int = PLC DIx_DB.T1_QF.Filter_Off.SP AT %DB9.DBW132, 1 s
   "T2_QF_Input" : Bool = PLC DIx_DB.T2_QF.Input AT %DB9.DBX140.0, 1 s
   "T2_QF_Signal" : Bool = PLC DIx_DB.T2_QF.Signal AT %DB9.DBX142.0, 1 s
   "T2_QF_Hand" : Bool = PLC DIx_DB.T2_QF.Hand AT %DB9.DBX144.0, 1 s
   "T2_QF_Start_M" : Bool = PLC DIx_DB.T2_QF.Start_M AT %DB9.DBX144.1, 1 s
   "T2_QF_Inverse" : Bool = PLC DIx_DB.T2_QF.Inverse AT %DB9.DBX144.3, 1 s
   "T2_QF_Filter_On_SP" : Int = PLC DIx_DB.T2_QF.Filter_On.SP AT %DB9.DBW146, 1 s
   "T2_QF_Filter_Off_SP" : Int = PLC DIx_DB.T2_QF.Filter_Off.SP AT %DB9.DBW152, 1 s
   "T3_QF_Input" : Bool = PLC DIx_DB.T3_QF.Input AT %DB9.DBX160.0, 1 s
   "T3_QF_Signal" : Bool = PLC DIx_DB.T3_QF.Signal AT %DB9.DBX162.0, 1 s
   "T3_QF_Hand" : Bool = PLC DIx_DB.T3_QF.Hand AT %DB9.DBX164.0, 1 s
   "T3_QF_Start_M" : Bool = PLC DIx_DB.T3_QF.Start_M AT %DB9.DBX164.1, 1 s
   "T3_QF_Inverse" : Bool = PLC DIx_DB.T3_QF.Inverse AT %DB9.DBX164.3, 1 s
   "T3_QF_Filter_On_SP" : Int = PLC DIx_DB.T3_QF.Filter_On.SP AT %DB9.DBW166, 1 s
   "T3_QF_Filter_Off_SP" : Int = PLC DIx_DB.T3_QF.Filter_Off.SP AT %DB9.DBW172, 1 s
   "T1_Box_ready_Input" : Bool = PLC DIx_DB.T1_Box_ready.Input AT %DB9.DBX180.0, 1 s
   "T1_Box_ready_Signal" : Bool = PLC DIx_DB.T1_Box_ready.Signal AT %DB9.DBX182.0, 1 s
   "T1_Box_ready_Hand" : Bool = PLC DIx_DB.T1_Box_ready.Hand AT %DB9.DBX184.0, 1 s
   "T1_Box_ready_Start_M" : Bool = PLC DIx_DB.T1_Box_ready.Start_M AT %DB9.DBX184.1, 1 s
   "T1_Box_ready_Inverse" : Bool = PLC DIx_DB.T1_Box_ready.Inverse AT %DB9.DBX184.3, 1 s
   "T1_Box_ready_Filter_On_SP" : Int = PLC DIx_DB.T1_Box_ready.Filter_On.SP AT %DB9.DBW186, 1 s
   "T1_Box_ready_Filter_Off_SP" : Int = PLC DIx_DB.T1_Box_ready.Filter_Off.SP AT %DB9.DBW192, 1 s
   "Air_pressure_Ok_Input" : Bool = PLC DIx_DB.Air_pressure_Ok.Input AT %DB9.DBX240.0, 1 s
   "Air_pressure_Ok_Signal" : Bool = PLC DIx_DB.Air_pressure_Ok.Signal AT %DB9.DBX242.0, 1 s
   "Air_pressure_Ok_Hand" : Bool = PLC DIx_DB.Air_pressure_Ok.Hand AT %DB9.DBX244.0, 1 s
   "Air_pressure_Ok_Start_M" : Bool = PLC DIx_DB.Air_pressure_Ok.Start_M AT %DB9.DBX244.1, 1 s
   "Air_pressure_Ok_Inverse" : Bool = PLC DIx_DB.Air_pressure_Ok.Inverse AT %DB9.DBX244.3, 1 s
   "Air_pressure_Ok_Filter_On_SP" : Int = PLC DIx_DB.Air_pressure_Ok.Filter_On.SP AT %DB9.DBW246, 1 s
   "Air_pressure_Ok_Filter_Off_SP" : Int = PLC DIx_DB.Air_pressure_Ok.Filter_Off.SP AT %DB9.DBW252, 1 s
   "T2_Box_Ready_Input" : Bool = PLC DIx_DB.T2_Box_Ready.Input AT %DB9.DBX200.0, 1 s
   "T2_Box_Ready_Signal" : Bool = PLC DIx_DB.T2_Box_Ready.Signal AT %DB9.DBX202.0, 1 s
   "T2_Box_Ready_Hand" : Bool = PLC DIx_DB.T2_Box_Ready.Hand AT %DB9.DBX204.0, 1 s
   "T2_Box_Ready_Start_M" : Bool = PLC DIx_DB.T2_Box_Ready.Start_M AT %DB9.DBX204.1, 1 s
   "T2_Box_Ready_Inverse" : Bool = PLC DIx_DB.T2_Box_Ready.Inverse AT %DB9.DBX204.3, 1 s
   "T2_Box_Ready_Filter_On_SP" : Int = PLC DIx_DB.T2_Box_Ready.Filter_On.SP AT %DB9.DBW206, 1 s
   "T2_Box_Ready_Filter_Off_SP" : Int = PLC DIx_DB.T2_Box_Ready.Filter_Off.SP AT %DB9.DBW212, 1 s
   "T3_Box_Ready_Hand" : Bool = PLC DIx_DB.T3_Box_Ready.Hand AT %DB9.DBX224.0, 1 s
   "T3_Box_Ready_Start_M" : Bool = PLC DIx_DB.T3_Box_Ready.Start_M AT %DB9.DBX224.1, 1 s
   "T3_Box_Ready_Inverse" : Bool = PLC DIx_DB.T3_Box_Ready.Inverse AT %DB9.DBX224.3, 1 s
   "T3_Box_Ready_Filter_On_SP" : Int = PLC DIx_DB.T3_Box_Ready.Filter_On.SP AT %DB9.DBW226, 1 s
   "T3_Box_Ready_Filter_Off_SP" : Int = PLC DIx_DB.T3_Box_Ready.Filter_Off.SP AT %DB9.DBW232, 1 s
   "FB_K1_Close_Input" : Bool = PLC DIx_DB.FB_K1_Close.Input AT %DB9.DBX260.0, 1 s
   "FB_K1_Close_Signal" : Bool = PLC DIx_DB.FB_K1_Close.Signal AT %DB9.DBX262.0, 1 s
   "FB_K1_Close_Hand" : Bool = PLC DIx_DB.FB_K1_Close.Hand AT %DB9.DBX264.0, 1 s
   "FB_K1_Close_Start_M" : Bool = PLC DIx_DB.FB_K1_Close.Start_M AT %DB9.DBX264.1, 1 s
   "FB_K1_Close_Inverse" : Bool = PLC DIx_DB.FB_K1_Close.Inverse AT %DB9.DBX264.3, 1 s
   "FB_K1_Close_Filter_On_SP" : Int = PLC DIx_DB.FB_K1_Close.Filter_On.SP AT %DB9.DBW266, 1 s
   "FB_K1_Close_Filter_Off_SP" : Int = PLC DIx_DB.FB_K1_Close.Filter_Off.SP AT %DB9.DBW272, 1 s
   "FB_K2_Open_Input" : Bool = PLC DIx_DB.FB_K2_Open.Input AT %DB9.DBX280.0, 1 s
   "FB_K2_Open_Signal" : Bool = PLC DIx_DB.FB_K2_Open.Signal AT %DB9.DBX282.0, 1 s
   "FB_K2_Open_Hand" : Bool = PLC DIx_DB.FB_K2_Open.Hand AT %DB9.DBX284.0, 1 s
   "FB_K2_Open_Start_M" : Bool = PLC DIx_DB.FB_K2_Open.Start_M AT %DB9.DBX284.1, 1 s
   "FB_K2_Open_Inverse" : Bool = PLC DIx_DB.FB_K2_Open.Inverse AT %DB9.DBX284.3, 1 s
   "FB_K2_Open_Filter_On_SP" : Int = PLC DIx_DB.FB_K2_Open.Filter_On.SP AT %DB9.DBW286, 1 s
   "FB_K2_Open_Filter_Off_SP" : Int = PLC DIx_DB.FB_K2_Open.Filter_Off.SP AT %DB9.DBW292, 1 s
   "FB_K2_Close_Input" : Bool = PLC DIx_DB.FB_K2_Close.Input AT %DB9.DBX300.0, 1 s
   "FB_K2_Close_Signal" : Bool = PLC DIx_DB.FB_K2_Close.Signal AT %DB9.DBX302.0, 1 s
   "FB_K2_Close_Hand" : Bool = PLC DIx_DB.FB_K2_Close.Hand AT %DB9.DBX304.0, 1 s
   "FB_K2_Close_Start_M" : Bool = PLC DIx_DB.FB_K2_Close.Start_M AT %DB9.DBX304.1, 1 s
   "FB_K2_Close_Inverse" : Bool = PLC DIx_DB.FB_K2_Close.Inverse AT %DB9.DBX304.3, 1 s
   "FB_K2_Close_Filter_On_SP" : Int = PLC DIx_DB.FB_K2_Close.Filter_On.SP AT %DB9.DBW306, 1 s
   "FB_K2_Close_Filter_Off_SP" : Int = PLC DIx_DB.FB_K2_Close.Filter_Off.SP AT %DB9.DBW312, 1 s
   "FB_K3_Open_Input" : Bool = PLC DIx_DB.FB_K3_Open.Input AT %DB9.DBX320.0, 1 s
   "FB_K3_Open_Signal" : Bool = PLC DIx_DB.FB_K3_Open.Signal AT %DB9.DBX322.0, 1 s
   "FB_K3_Open_Hand" : Bool = PLC DIx_DB.FB_K3_Open.Hand AT %DB9.DBX324.0, 1 s
   "FB_K3_Open_Start_M" : Bool = PLC DIx_DB.FB_K3_Open.Start_M AT %DB9.DBX324.1, 1 s
   "FB_K3_Open_Inverse" : Bool = PLC DIx_DB.FB_K3_Open.Inverse AT %DB9.DBX324.3, 1 s
   "FB_K3_Open_Filter_On_SP" : Int = PLC DIx_DB.FB_K3_Open.Filter_On.SP AT %DB9.DBW326, 1 s
   "FB_K3_Open_Filter_Off_SP" : Int = PLC DIx_DB.FB_K3_Open.Filter_Off.SP AT %DB9.DBW332, 1 s
   "FB_K3_Close_Input" : Bool = PLC DIx_DB.FB_K3_Close.Input AT %DB9.DBX340.0, 1 s
   "FB_K3_Close_Signal" : Bool = PLC DIx_DB.FB_K3_Close.Signal AT %DB9.DBX342.0, 1 s
   "FB_K3_Close_Hand" : Bool = PLC DIx_DB.FB_K3_Close.Hand AT %DB9.DBX344.0, 1 s
   "FB_K3_Close_Start_M" : Bool = PLC DIx_DB.FB_K3_Close.Start_M AT %DB9.DBX344.1, 1 s
   "FB_K3_Close_Inverse" : Bool = PLC DIx_DB.FB_K3_Close.Inverse AT %DB9.DBX344.3, 1 s
   "FB_K3_Close_Filter_Off_SP" : Int = PLC DIx_DB.FB_K3_Close.Filter_Off.SP AT %DB9.DBW352, 1 s
   "T3_Box_Ready_Signal" : Bool = PLC DIx_DB.T3_Box_Ready.Signal AT %DB9.DBX222.0, 1 s
   "FB_K3_Close_Filter_On_SP" : Int = PLC DIx_DB.FB_K3_Close.Filter_On.SP AT %DB9.DBW346, 1 s
   "T3_Box_Ready_Input" : Bool = PLC DIx_DB.T3_Box_Ready.Input AT %DB9.DBX220.0, 1 s

HMI tags "DOx"
   "ODT0_CMD_Start_A" : Bool = PLC DOx_DB.T0_CMD.Start AT %DB6.DBX0.0, 1 s
   "ODT0_CMD_Start_M" : Bool = PLC DOx_DB.T0_CMD.Start_M AT %DB6.DBX2.1, 1 s
   "ODT0_CMD_Q" : Bool = PLC DOx_DB.T0_CMD.Q AT %DB6.DBX0.2, 1 s
   "ODT0_CMD_Hand" : Bool = PLC DOx_DB.T0_CMD.Hand AT %DB6.DBX2.0, 1 s
   "ODT0_CMD_Inverse" : Bool = PLC DOx_DB.T0_CMD.Inverse AT %DB6.DBX2.3, 1 s
   "ODT0_CMD_Simulation" : Bool = PLC DOx_DB.T0_CMD.Simulation AT %DB6.DBX2.2, 1 s
   "ODT1_CMD_Start_A" : Bool = PLC DOx_DB.T1_CMD.Start_M AT %DB6.DBX12.1, 1 s
   "ODT1_CMD_Q" : Bool = PLC DOx_DB.T1_CMD.Q AT %DB6.DBX10.2, 1 s
   "ODT1_CMD_Hand" : Bool = PLC DOx_DB.T1_CMD.Hand AT %DB6.DBX12.0, 1 s
   "ODT1_CMD_Start_M" : Bool = PLC DOx_DB.T1_CMD.Start_M AT %DB6.DBX12.1, 1 s
   "ODT1_CMD_Simulation" : Bool = PLC DOx_DB.T1_CMD.Simulation AT %DB6.DBX12.2, 1 s
   "ODT1_CMD_Inverse" : Bool = PLC DOx_DB.T1_CMD.Inverse AT %DB6.DBX12.3, 1 s
   "ODT2_CMD_Start_A" : Bool = PLC DOx_DB.T2_CMD.Start AT %DB6.DBX20.0, 1 s
   "ODT2_CMD_Q" : Bool = PLC DOx_DB.T2_CMD.Q AT %DB6.DBX20.2, 1 s
   "ODT2_CMD_Hand" : Bool = PLC DOx_DB.T2_CMD.Hand AT %DB6.DBX22.0, 1 s
   "ODT2_CMD_Start_M" : Bool = PLC DOx_DB.T2_CMD.Start_M AT %DB6.DBX22.1, 1 s
   "ODT2_CMD_Simulation" : Bool = PLC DOx_DB.T2_CMD.Simulation AT %DB6.DBX22.2, 1 s
   "ODT2_CMD_Inverse" : Bool = PLC DOx_DB.T2_CMD.Inverse AT %DB6.DBX22.3, 1 s
   "ODT3_CMD_Start_A" : Bool = PLC DOx_DB.T3_CMD.Start AT %DB6.DBX30.0, 1 s
   "ODT3_CMD_Q" : Bool = PLC DOx_DB.T3_CMD.Q AT %DB6.DBX30.2, 1 s
   "ODT3_CMD_Hand" : Bool = PLC DOx_DB.T3_CMD.Hand AT %DB6.DBX32.0, 1 s
   "ODT3_CMD_Start_M" : Bool = PLC DOx_DB.T3_CMD.Start_M AT %DB6.DBX32.1, 1 s
   "ODT3_CMD_Simulation" : Bool = PLC DOx_DB.T3_CMD.Simulation AT %DB6.DBX32.2, 1 s
   "ODT3_CMD_Inverse" : Bool = PLC DOx_DB.T3_CMD.Inverse AT %DB6.DBX32.3, 1 s
   "K1_CMD_Start_A" : Bool = PLC DOx_DB.K1_CMD.Start AT %DB6.DBX40.0, 1 s
   "K1_CMD_Q" : Bool = PLC DOx_DB.K1_CMD.Q AT %DB6.DBX40.2, 1 s
   "K1_CMD_Hand" : Bool = PLC DOx_DB.K1_CMD.Hand AT %DB6.DBX42.0, 1 s
   "K1_CMD_Start_M" : Bool = PLC DOx_DB.K1_CMD.Start_M AT %DB6.DBX42.1, 1 s
   "K1_CMD_Simulation" : Bool = PLC DOx_DB.K1_CMD.Simulation AT %DB6.DBX42.2, 1 s
   "K1_CMD_Inverse" : Bool = PLC DOx_DB.K1_CMD.Inverse AT %DB6.DBX42.3, 1 s
   "K2_CMD_Start_A" : Bool = PLC DOx_DB.K2_CMD.Start AT %DB6.DBX50.0, 1 s
   "K2_CMD_Q" : Bool = PLC DOx_DB.K2_CMD.Q AT %DB6.DBX50.2, 1 s
   "K2_CMD_Hand" : Bool = PLC DOx_DB.K2_CMD.Hand AT %DB6.DBX52.0, 1 s
   "K2_CMD_Start_M" : Bool = PLC DOx_DB.K2_CMD.Start_M AT %DB6.DBX52.1, 1 s
   "K2_CMD_Simulation" : Bool = PLC DOx_DB.K2_CMD.Simulation AT %DB6.DBX52.2, 1 s
   "K2_CMD_Inverse" : Bool = PLC DOx_DB.K2_CMD.Inverse AT %DB6.DBX52.3, 1 s
   "K3_CMD_Start_A" : Bool = PLC DOx_DB.K3_CMD.Start AT %DB6.DBX60.0, 1 s
   "K3_CMD_Q" : Bool = PLC DOx_DB.K3_CMD.Q AT %DB6.DBX60.2, 1 s
   "K3_CMD_Hand" : Bool = PLC DOx_DB.K3_CMD.Hand AT %DB6.DBX62.0, 1 s
   "K3_CMD_Start_M" : Bool = PLC DOx_DB.K3_CMD.Start_M AT %DB6.DBX62.1, 1 s
   "K3_CMD_Simulation" : Bool = PLC DOx_DB.K3_CMD.Simulation AT %DB6.DBX62.2, 1 s
   "K3_CMD_Inverse" : Bool = PLC DOx_DB.K3_CMD.Inverse AT %DB6.DBX62.3, 1 s
   "Supply_allowed_Start_A" : Bool = PLC DOx_DB.Supply_allowed.Start AT %DB6.DBX70.0, 1 s
   "Supply_allowed_Q" : Bool = PLC DOx_DB.Supply_allowed.Q AT %DB6.DBX70.2, 1 s
   "Supply_allowed_Hand" : Bool = PLC DOx_DB.Supply_allowed.Hand AT %DB6.DBX72.0, 1 s
   "Supply_allowed_Start_M" : Bool = PLC DOx_DB.Supply_allowed.Start_M AT %DB6.DBX72.1, 1 s
   "Supply_allowed_Simulation" : Bool = PLC DOx_DB.Supply_allowed.Simulation AT %DB6.DBX72.2, 1 s
   "Supply_allowed_Inverse" : Bool = PLC DOx_DB.Supply_allowed.Inverse AT %DB6.DBX72.3, 1 s
   "Reset_Safety_Start_A" : Bool = PLC DOx_DB.Reset_Safety.Start AT %DB6.DBX80.0, 1 s
   "Reset_Safety_Q" : Bool = PLC DOx_DB.Reset_Safety.Q AT %DB6.DBX80.2, 1 s
   "Reset_Safety_Hand" : Bool = PLC DOx_DB.Reset_Safety.Hand AT %DB6.DBX82.0, 1 s
   "Reset_Safety_Start_M" : Bool = PLC DOx_DB.Reset_Safety.Start_M AT %DB6.DBX82.1, 1 s
   "Reset_Safety_Simulation" : Bool = PLC DOx_DB.Reset_Safety.Simulation AT %DB6.DBX82.2, 1 s
   "Reset_Safety_Inverse" : Bool = PLC DOx_DB.Reset_Safety.Inverse AT %DB6.DBX82.3, 1 s
   "Reset_Start_A" : Bool = PLC DOx_DB.Reset.Start AT %DB6.DBX90.0, 1 s
   "Reset_Q" : Bool = PLC DOx_DB.Reset.Q AT %DB6.DBX90.2, 1 s
   "Reset_Hand" : Bool = PLC DOx_DB.Reset.Hand AT %DB6.DBX92.0, 1 s
   "Reset_Start_M" : Bool = PLC DOx_DB.Reset.Start_M AT %DB6.DBX92.1, 1 s
   "Reset_Simulation" : Bool = PLC DOx_DB.Reset.Simulation AT %DB6.DBX92.2, 1 s
   "Reset_Inverse" : Bool = PLC DOx_DB.Reset.Inverse AT %DB6.DBX92.3, 1 s
   "Green_Start_A" : Bool = PLC DOx_DB.Green.Start AT %DB6.DBX100.0, 1 s
   "Green_Q" : Bool = PLC DOx_DB.Green.Q AT %DB6.DBX100.2, 1 s
   "Green_Hand" : Bool = PLC DOx_DB.Green.Hand AT %DB6.DBX102.0, 1 s
   "Green_Start_M" : Bool = PLC DOx_DB.Green.Start_M AT %DB6.DBX102.1, 1 s
   "Green_Simulation" : Bool = PLC DOx_DB.Green.Simulation AT %DB6.DBX102.2, 1 s
   "Green_Inverse" : Bool = PLC DOx_DB.Green.Inverse AT %DB6.DBX102.3, 1 s
   "Red_Start_A" : Bool = PLC DOx_DB.Red.Start AT %DB6.DBX110.0, 1 s
   "Red_Q" : Bool = PLC DOx_DB.Red.Q AT %DB6.DBX110.2, 1 s
   "Red_Hand" : Bool = PLC DOx_DB.Red.Hand AT %DB6.DBX112.0, 1 s
   "Red_Start_M" : Bool = PLC DOx_DB.Red.Start_M AT %DB6.DBX112.1, 1 s
   "Red_Simulation" : Bool = PLC DOx_DB.Red.Simulation AT %DB6.DBX112.2, 1 s
   "Red_Inverse" : Bool = PLC DOx_DB.Red.Inverse AT %DB6.DBX112.3, 1 s
   "Blue_Start_A" : Bool = PLC DOx_DB.Blue.Start AT %DB6.DBX120.0, 1 s
   "Blue_Q" : Bool = PLC DOx_DB.Blue.Q AT %DB6.DBX120.2, 1 s
   "Blue_Hand" : Bool = PLC DOx_DB.Blue.Hand AT %DB6.DBX122.0, 1 s
   "Blue_Start_M" : Bool = PLC DOx_DB.Blue.Start_M AT %DB6.DBX122.1, 1 s
   "Blue_Simulation" : Bool = PLC DOx_DB.Blue.Simulation AT %DB6.DBX122.2, 1 s
   "Blue_Inverse" : Bool = PLC DOx_DB.Blue.Inverse AT %DB6.DBX122.3, 1 s
   "Orange_Start_A" : Bool = PLC DOx_DB.Orange.Start_M AT %DB6.DBX132.1, 1 s
   "Orange_Q" : Bool = PLC DOx_DB.Orange.Q AT %DB6.DBX130.2, 1 s
   "Orange_Hand" : Bool = PLC DOx_DB.Orange.Hand AT %DB6.DBX132.0, 1 s
   "Orange_Start_M" : Bool = PLC DOx_DB.Orange.Start_M AT %DB6.DBX132.1, 1 s
   "Orange_Simulation" : Bool = PLC DOx_DB.Orange.Simulation AT %DB6.DBX132.2, 1 s
   "Orange_Inverse" : Bool = PLC DOx_DB.Orange.Inverse AT %DB6.DBX132.3, 1 s

HMI tags "SP"
   "T4D4_S2_SP" : Real = PLC T4D4_DB.S2.SP AT %DB10.DBD24, 1 s
   "T4D4_DB_S2_Now" : Real = PLC T4D4_DB.S2.Now AT %DB10.DBD28, 1 s
   "Sp_view" : Int AT %DB1.DBD0

HMI tags "statistic"
   "b_1" : Int = PLC Statistic_DB.move_stat_Instance.box[1] AT %DB19.DBW102, 1 s
   "b_2" : Int = PLC Statistic_DB.move_stat_Instance.box[2] AT %DB19.DBW104, 1 s
   "b_3" : Int = PLC Statistic_DB.move_stat_Instance.box[3] AT %DB19.DBW106, 1 s
   "b_4" : Int = PLC Statistic_DB.move_stat_Instance.box[4] AT %DB19.DBW108, 1 s
   "b_5" : Int = PLC Statistic_DB.move_stat_Instance.box[5] AT %DB19.DBW110, 1 s
   "b_6" : Int = PLC Statistic_DB.move_stat_Instance.box[6] AT %DB19.DBW112, 1 s
   "b_7" : Int = PLC Statistic_DB.move_stat_Instance.box[7] AT %DB19.DBW114, 1 s
   "b_8" : Int = PLC Statistic_DB.move_stat_Instance.box[8] AT %DB19.DBW116, 1 s
   "b_9" : Int = PLC Statistic_DB.move_stat_Instance.box[9] AT %DB19.DBW118, 1 s
   "b_10" : Int = PLC Statistic_DB.move_stat_Instance.box[10] AT %DB19.DBW120, 1 s
   "b_11" : Int = PLC Statistic_DB.move_stat_Instance.box[11] AT %DB19.DBW122, 1 s
   "b_12" : Int = PLC Statistic_DB.move_stat_Instance.box[12] AT %DB19.DBW124, 1 s
   "b_13" : Int = PLC Statistic_DB.move_stat_Instance.box[13] AT %DB19.DBW126, 1 s
   "b_14" : Int = PLC Statistic_DB.move_stat_Instance.box[14] AT %DB19.DBW128, 1 s
   "b_15" : Int = PLC Statistic_DB.move_stat_Instance.box[15] AT %DB19.DBW130, 1 s
   "b_16" : Int = PLC Statistic_DB.move_stat_Instance.box[16] AT %DB19.DBW132, 1 s
   "b_17" : Int = PLC Statistic_DB.move_stat_Instance.box[17] AT %DB19.DBW134, 1 s
   "b_18" : Int = PLC Statistic_DB.move_stat_Instance.box[18] AT %DB19.DBW136, 1 s
   "b_19" : Int = PLC Statistic_DB.move_stat_Instance.box[19] AT %DB19.DBW138, 1 s
   "b_20" : Int = PLC Statistic_DB.move_stat_Instance.box[20] AT %DB19.DBW140, 1 s
   "b_21" : Int = PLC Statistic_DB.move_stat_Instance.box[21] AT %DB19.DBW142, 1 s
   "b_22" : Int = PLC Statistic_DB.move_stat_Instance.box[22] AT %DB19.DBW144, 1 s
   "b_23" : Int = PLC Statistic_DB.move_stat_Instance.box[23] AT %DB19.DBW146, 1 s
   "b_24" : Int = PLC Statistic_DB.move_stat_Instance.box[24] AT %DB19.DBW148, 1 s
   "b_25" : Int = PLC Statistic_DB.move_stat_Instance.box[25] AT %DB19.DBW150, 1 s

HMI tags "Standard-Variablentabelle"
   "WP231PR_DB_DR03_RESERVED_130" : String[12] = PLC WP231PR_DB.DR03.RESERVED_130 AT %DB231.DBX662.0, 1 s

HMI tags "Data Record DR3"
   "WP231PR_DB_DR03_SCALE_NAME" : String[12] = PLC WP231PR_DB.DR03.SCALE_NAME AT %DB231.DBX542.0, 1 s
   "WP231PR_DB_DR03_WEIGHT_UNIT" : String[4] = PLC WP231PR_DB.DR03.WEIGHT_UNIT AT %DB231.DBX556.0, 1 s
   "WP231PR_DB_DR03_LETTER_GROSS_WEIGHT_2" : Byte = PLC WP231PR_DB.DR03.LETTER_GROSS_WEIGHT_2 AT %DB231.DBB565, 1 s
   "WP231PR_DB_DR03_RESTRICTION_CODE" : UInt = PLC WP231PR_DB.DR03.RESTRICTION_CODE AT %DB231.DBW568, 1 s
   "WP231PR_DB_DR03_MIN_WEIGHT_D" : UInt = PLC WP231PR_DB.DR03.MIN_WEIGHT_D AT %DB231.DBW570, 1 s
   "WP231PR_DB_DR03_MAX_WEIGHT" : Real = PLC WP231PR_DB.DR03.MAX_WEIGHT AT %DB231.DBD574, 1 s
   "WP231PR_DB_DR03_CALIB_WEIGHT_0" : Real = PLC WP231PR_DB.DR03.CALIB_WEIGHT_0 AT %DB231.DBD578, 1 s
   "WP231PR_DB_DR03_CALIB_WEIGHT_1" : Real = PLC WP231PR_DB.DR03.CALIB_WEIGHT_1 AT %DB231.DBD582, 1 s
   "WP231PR_DB_DR03_CALIB_WEIGHT_2" : Real = PLC WP231PR_DB.DR03.CALIB_WEIGHT_2 AT %DB231.DBD586, 1 s
   "WP231PR_DB_DR03_CALIB_DIGITS_0" : DInt = PLC WP231PR_DB.DR03.CALIB_DIGITS_0 AT %DB231.DBD590, 1 s
   "WP231PR_DB_DR03_CALIB_DIGITS_1" : DInt = PLC WP231PR_DB.DR03.CALIB_DIGITS_1 AT %DB231.DBD594, 1 s
   "WP231PR_DB_DR03_CALIB_DIGITS_2" : DInt = PLC WP231PR_DB.DR03.CALIB_DIGITS_2 AT %DB231.DBD598, 1 s
   "WP231PR_DB_DR03_RESOLUTION_D" : Real = PLC WP231PR_DB.DR03.RESOLUTION_D AT %DB231.DBD602, 1 s
   "WP231PR_DB_DR03_INITIAL_ZEROING" : Bool = PLC WP231PR_DB.DR03.INITIAL_ZEROING AT %DB231.DBX607.0, 1 s
   "WP231PR_DB_DR03_INITIAL_ZEROING_IF_TARED" : Bool = PLC WP231PR_DB.DR03.INITIAL_ZEROING_IF_TARED AT %DB231.DBX607.1, 1 s
   "WP231PR_DB_DR03_ZERO_TRACKING" : Bool = PLC WP231PR_DB.DR03.ZERO_TRACKING AT %DB231.DBX607.2, 1 s
   "WP231PR_DB_DR03_ADDITIVE_TARE" : Bool = PLC WP231PR_DB.DR03.ADDITIVE_TARE AT %DB231.DBX607.3, 1 s
   "WP231PR_DB_DR03_WEIGHT_SIM_ALLOWED" : Bool = PLC WP231PR_DB.DR03.WEIGHT_SIM_ALLOWED AT %DB231.DBX607.4, 1 s
   "WP231PR_DB_DR03_DEC_POINT_PROC_VAL" : UInt = PLC WP231PR_DB.DR03.DEC_POINT_PROC_VAL AT %DB231.DBW608, 1 s
   "WP231PR_DB_DR03_TARE_MAX" : Real = PLC WP231PR_DB.DR03.TARE_MAX AT %DB231.DBD610, 1 s
   "WP231PR_DB_DR03_INITIAL_ZEROING_LIM_NEG" : Real = PLC WP231PR_DB.DR03.INITIAL_ZEROING_LIM_NEG AT %DB231.DBD614, 1 s
   "WP231PR_DB_DR03_INITIAL_ZEROING_LIM_POS" : Real = PLC WP231PR_DB.DR03.INITIAL_ZEROING_LIM_POS AT %DB231.DBD618, 1 s
   "WP231PR_DB_DR03_SEM_AUT_ZERO_LIM_NEG" : Real = PLC WP231PR_DB.DR03.SEM_AUT_ZERO_LIM_NEG AT %DB231.DBD622, 1 s
   "WP231PR_DB_DR03_SEM_AUT_ZERO_LIM_POS" : Real = PLC WP231PR_DB.DR03.SEM_AUT_ZERO_LIM_POS AT %DB231.DBD626, 1 s
   "WP231PR_DB_DR03_ST_STILL_RANGE_D" : Real = PLC WP231PR_DB.DR03.ST_STILL_RANGE_D AT %DB231.DBD630, 1 s
   "WP231PR_DB_DR03_ST_STILL_TIME" : Time = PLC WP231PR_DB.DR03.ST_STILL_TIME AT %DB231.DBD634, 1 s
   "WP231PR_DB_DR03_ST_STILL_WAITING_TIME" : Time = PLC WP231PR_DB.DR03.ST_STILL_WAITING_TIME AT %DB231.DBD638, 1 s
   "WP231PR_DB_DR03_FREQ_LOW_PASS_1" : Real = PLC WP231PR_DB.DR03.FREQ_LOW_PASS_1 AT %DB231.DBD642, 1 s
   "WP231PR_DB_DR03_ORDER_NO_LOW_PASS_1" : UInt = PLC WP231PR_DB.DR03.ORDER_NO_LOW_PASS_1 AT %DB231.DBW646, 1 s
   "WP231PR_DB_DR03_FREQ_LOW_PASS_2" : Real = PLC WP231PR_DB.DR03.FREQ_LOW_PASS_2 AT %DB231.DBD650, 1 s
   "WP231PR_DB_DR03_ORDER_NO_LOW_PASS_2" : UInt = PLC WP231PR_DB.DR03.ORDER_NO_LOW_PASS_2 AT %DB231.DBW654, 1 s
   "WP231PR_DB_DR03_AVER_FILTER_DEPTH" : UInt = PLC WP231PR_DB.DR03.AVER_FILTER_DEPTH AT %DB231.DBW656, 1 s
   "WP231PR_DB_DR03_SHOW_WR_DATA" : UInt = PLC WP231PR_DB.DR03.SHOW_WR_DATA AT %DB231.DBW658, 1 s
   "WP231PR_DB_DR03_SECURE_DISPLAY_INTERFACE" : UInt = PLC WP231PR_DB.DR03.SECURE_DISPLAY_INTERFACE AT %DB231.DBW660, 1 s
   "WP231PR_DB_DR03_FW_VERSION_HMI_MODUL" : String[20] = PLC WP231PR_DB.DR03.FW_VERSION_HMI_MODUL AT %DB231.DBX698.0, 1 s
   "WP231PR_DB_DR03_MIN_ZOOMFACTOR" : UInt = PLC WP231PR_DB.DR03.MIN_ZOOMFACTOR AT %DB231.DBW720, 1 s

HMI tags "Data Record DR4"
   "WP231PR_DB_DR04_CALIB_DIGITS_0_CALC" : DInt = PLC WP231PR_DB.DR04.CALIB_DIGITS_0_CALC AT %DB231.DBD734, 1 s
   "WP231PR_DB_DR04_CALIB_DIGITS_1_CALC" : DInt = PLC WP231PR_DB.DR04.CALIB_DIGITS_1_CALC AT %DB231.DBD738, 1 s
   "WP231PR_DB_DR04_CALIB_DIGITS_2_CALC" : DInt = PLC WP231PR_DB.DR04.CALIB_DIGITS_2_CALC AT %DB231.DBD742, 1 s

HMI tags "Data Record DR5"
   "WP231PR_DB_DR05_TARE_WEIGHT_PRESET" : Real = PLC WP231PR_DB.DR05.TARE_WEIGHT_PRESET AT %DB231.DBD762, 1 s
   "WP231PR_DB_DR05_TARE_WEIGHT_SEM_AUT" : Real = PLC WP231PR_DB.DR05.TARE_WEIGHT_SEM_AUT AT %DB231.DBD766, 1 s
   "WP231PR_DB_DR05_ZEROING_WEIGHT_INITIAL" : Real = PLC WP231PR_DB.DR05.ZEROING_WEIGHT_INITIAL AT %DB231.DBD770, 1 s
   "WP231PR_DB_DR05_ZEROING_WEIGHT_SEM_AUT" : Real = PLC WP231PR_DB.DR05.ZEROING_WEIGHT_SEM_AUT AT %DB231.DBD774, 1 s
   "WP231PR_DB_DR05_ZEROING_WEIGHT_TRACKING" : Real = PLC WP231PR_DB.DR05.ZEROING_WEIGHT_TRACKING AT %DB231.DBD778, 1 s
   "WP231PR_DB_DR05_DEAD_LOAD" : Real = PLC WP231PR_DB.DR05.DEAD_LOAD AT %DB231.DBD782, 1 s

HMI tags "Data Record DR6"
   "WP231PR_DB_DR06_LIM_REFERENCE" : UInt = PLC WP231PR_DB.DR06.LIM_REFERENCE AT %DB231.DBW802, 1 s
   "WP231PR_DB_DR06_LIM_1_ON" : Real = PLC WP231PR_DB.DR06.LIM_1_ON AT %DB231.DBD806, 1 s
   "WP231PR_DB_DR06_DELAY_LIM_1_ON" : Time = PLC WP231PR_DB.DR06.DELAY_LIM_1_ON AT %DB231.DBD810, 1 s
   "WP231PR_DB_DR06_LIM_1_OFF" : Real = PLC WP231PR_DB.DR06.LIM_1_OFF AT %DB231.DBD814, 1 s
   "WP231PR_DB_DR06_DELAY_LIM_1_OFF" : Time = PLC WP231PR_DB.DR06.DELAY_LIM_1_OFF AT %DB231.DBD818, 1 s
   "WP231PR_DB_DR06_LIM_2_ON" : Real = PLC WP231PR_DB.DR06.LIM_2_ON AT %DB231.DBD822, 1 s
   "WP231PR_DB_DR06_DELAY_LIM_2_ON" : Time = PLC WP231PR_DB.DR06.DELAY_LIM_2_ON AT %DB231.DBD826, 1 s
   "WP231PR_DB_DR06_LIM_2_OFF" : Real = PLC WP231PR_DB.DR06.LIM_2_OFF AT %DB231.DBD830, 1 s
   "WP231PR_DB_DR06_DELAY_LIM_2_OFF" : Time = PLC WP231PR_DB.DR06.DELAY_LIM_2_OFF AT %DB231.DBD834, 1 s
   "WP231PR_DB_DR06_LIMIT_3_EMPTY" : Real = PLC WP231PR_DB.DR06.LIMIT_3_EMPTY AT %DB231.DBD838, 1 s
   "WP231PR_DB_DR06_DELAY_EMPTY" : Time = PLC WP231PR_DB.DR06.DELAY_EMPTY AT %DB231.DBD842, 1 s

HMI tags "Data Record DR7"
   "WP231PR_DB_DR07_ASSIGN_DI_0" : UInt = PLC WP231PR_DB.DR07.ASSIGN_DI_0 AT %DB231.DBW862, 1 s
   "WP231PR_DB_DR07_ASSIGN_DI_1" : UInt = PLC WP231PR_DB.DR07.ASSIGN_DI_1 AT %DB231.DBW864, 1 s
   "WP231PR_DB_DR07_ASSIGN_DI_2" : UInt = PLC WP231PR_DB.DR07.ASSIGN_DI_2 AT %DB231.DBW866, 1 s
   "WP231PR_DB_DR07_ASSIGN_DI_3" : UInt = PLC WP231PR_DB.DR07.ASSIGN_DI_3 AT %DB231.DBW868, 1 s
   "WP231PR_DB_DR07_FILTER_DI" : UInt = PLC WP231PR_DB.DR07.FILTER_DI AT %DB231.DBW870, 1 s
   "WP231PR_DB_DR07_ASSIGN_DQ_0" : UInt = PLC WP231PR_DB.DR07.ASSIGN_DQ_0 AT %DB231.DBW872, 1 s
   "WP231PR_DB_DR07_ASSIGN_DQ_1" : UInt = PLC WP231PR_DB.DR07.ASSIGN_DQ_1 AT %DB231.DBW874, 1 s
   "WP231PR_DB_DR07_ASSIGN_DQ_2" : UInt = PLC WP231PR_DB.DR07.ASSIGN_DQ_2 AT %DB231.DBW876, 1 s
   "WP231PR_DB_DR07_ASSIGN_DQ_3" : UInt = PLC WP231PR_DB.DR07.ASSIGN_DQ_3 AT %DB231.DBW878, 1 s
   "WP231PR_DB_DR07_ANA_OUT_BY_ERR_OR_STOP" : UInt = PLC WP231PR_DB.DR07.ANA_OUT_BY_ERR_OR_STOP AT %DB231.DBW880, 1 s
   "WP231PR_DB_DR07_DQ_0_BY_ERR_OR_STOP" : Bool = PLC WP231PR_DB.DR07.DQ_0_BY_ERR_OR_STOP AT %DB231.DBX883.0, 1 s
   "WP231PR_DB_DR07_DQ_1_BY_ERR_OR_STOP" : Bool = PLC WP231PR_DB.DR07.DQ_1_BY_ERR_OR_STOP AT %DB231.DBX883.1, 1 s
   "WP231PR_DB_DR07_DQ_2_BY_ERR_OR_STOP" : Bool = PLC WP231PR_DB.DR07.DQ_2_BY_ERR_OR_STOP AT %DB231.DBX883.2, 1 s
   "WP231PR_DB_DR07_DQ_3_BY_ERR_OR_STOP" : Bool = PLC WP231PR_DB.DR07.DQ_3_BY_ERR_OR_STOP AT %DB231.DBX883.3, 1 s
   "WP231PR_DB_DR07_RANGE_ANA_OUT" : UInt = PLC WP231PR_DB.DR07.RANGE_ANA_OUT AT %DB231.DBW884, 1 s
   "WP231PR_DB_DR07_SOURCE_ANA_OUT" : UInt = PLC WP231PR_DB.DR07.SOURCE_ANA_OUT AT %DB231.DBW886, 1 s
   "WP231PR_DB_DR07_ANA_OUT_BY_ERR_OR_STOP_1" : UInt = PLC WP231PR_DB.DR07.ANA_OUT_BY_ERR_OR_STOP_1 AT %DB231.DBW888, 1 s
   "WP231PR_DB_DR07_START_VAL_ANA_OUT" : Real = PLC WP231PR_DB.DR07.START_VAL_ANA_OUT AT %DB231.DBD890, 1 s
   "WP231PR_DB_DR07_END_VAL_ANA_OUT" : Real = PLC WP231PR_DB.DR07.END_VAL_ANA_OUT AT %DB231.DBD894, 1 s
   "WP231PR_DB_DR07_ANA_OUT_ERR" : Real = PLC WP231PR_DB.DR07.ANA_OUT_ERR AT %DB231.DBD898, 1 s
   "WP231PR_DB_DR07_TRACE_RATE" : UInt = PLC WP231PR_DB.DR07.TRACE_RATE AT %DB231.DBW902, 1 s
   "WP231PR_DB_DR07_TRACE_MEM_TYPE" : Bool = PLC WP231PR_DB.DR07.TRACE_MEM_TYPE AT %DB231.DBX905.0, 1 s

HMI tags "Data Record DR8"
   "WP231PR_DB_DR08_DATE_TIME" : DTL = PLC WP231PR_DB.DR08.DATE_TIME AT %DB231.DBX922.0, 1 s

HMI tags "Data Record DR9"
   "WP231PR_DB_DR09_ORDER_NO" : String[16] = PLC WP231PR_DB.DR09.ORDER_NO AT %DB231.DBX942.0, 1 s
   "WP231PR_DB_DR09_SERIAL_NO" : String[12] = PLC WP231PR_DB.DR09.SERIAL_NO AT %DB231.DBX960.0, 1 s
   "WP231PR_DB_DR09_FIRMWARE_VERS" : String[2] = PLC WP231PR_DB.DR09.FIRMWARE_VERS AT %DB231.DBX974.0, 1 s
   "WP231PR_DB_DR09_FIRMWARE_VERS_POS_1" : UInt = PLC WP231PR_DB.DR09.FIRMWARE_VERS_POS_1 AT %DB231.DBW978, 1 s
   "WP231PR_DB_DR09_FIRMWARE_VERS_POS_2" : UInt = PLC WP231PR_DB.DR09.FIRMWARE_VERS_POS_2 AT %DB231.DBW980, 1 s
   "WP231PR_DB_DR09_FIRMWARE_VERS_POS_3" : UInt = PLC WP231PR_DB.DR09.FIRMWARE_VERS_POS_3 AT %DB231.DBW982, 1 s
   "WP231PR_DB_DR09_HARDWARE_VERSION" : UInt = PLC WP231PR_DB.DR09.HARDWARE_VERSION AT %DB231.DBW984, 1 s
   "WP231PR_DB_DR09_OS_VERSION_2" : String[2] = PLC WP231PR_DB.DR09.OS_VERSION_2 AT %DB231.DBX986.0, 1 s
   "WP231PR_DB_DR09_OS_VERSION_1" : UInt = PLC WP231PR_DB.DR09.OS_VERSION_1 AT %DB231.DBW990, 1 s
   "WP231PR_DB_DR09_DRAM" : UInt = PLC WP231PR_DB.DR09.DRAM AT %DB231.DBW992, 1 s
   "WP231PR_DB_DR09_FLASH" : UInt = PLC WP231PR_DB.DR09.FLASH AT %DB231.DBW994, 1 s
   "WP231PR_DB_DR09_MRAM" : UInt = PLC WP231PR_DB.DR09.MRAM AT %DB231.DBW996, 1 s

HMI tags "Data Record DR10"
   "WP231PR_DB_DR10_NO_OF_LOAD_CELLS" : UInt = PLC WP231PR_DB.DR10.NO_OF_LOAD_CELLS AT %DB231.DBW1010, 1 s
   "WP231PR_DB_DR10_SWITCH_50_60_HZ" : UInt = PLC WP231PR_DB.DR10.SWITCH_50_60_HZ AT %DB231.DBW1012, 1 s
   "WP231PR_DB_DR10_NO_POINTS_OF_SUPPORT" : UInt = PLC WP231PR_DB.DR10.NO_POINTS_OF_SUPPORT AT %DB231.DBW1014, 1 s
   "WP231PR_DB_DR10_GAIN_LOAD_CELL" : Real = PLC WP231PR_DB.DR10.GAIN_LOAD_CELL AT %DB231.DBD1018, 1 s
   "WP231PR_DB_DR10_ZERO_OFFSET_LC" : Real = PLC WP231PR_DB.DR10.ZERO_OFFSET_LC AT %DB231.DBD1022, 1 s
   "WP231PR_DB_DR10_NOM_LOAD_ONE_LOAD_CELL" : Real = PLC WP231PR_DB.DR10.NOM_LOAD_ONE_LOAD_CELL AT %DB231.DBD1026, 1 s

HMI tags "Data Record DR12"
   "WP231PR_DB_DR12_DEVICE_MAC_ADDRESS" : UInt = PLC WP231PR_DB.DR12.DEVICE_MAC_ADDRESS AT %DB231.DBW1054, 1 s
   "WP231PR_DB_DR12_DEVICE_MAC_ADDRESS_1" : UInt = PLC WP231PR_DB.DR12.DEVICE_MAC_ADDRESS_1 AT %DB231.DBW1056, 1 s
   "WP231PR_DB_DR12_DEVICE_MAC_ADDRESS_2" : UInt = PLC WP231PR_DB.DR12.DEVICE_MAC_ADDRESS_2 AT %DB231.DBW1058, 1 s
   "WP231PR_DB_DR12_DEVICE_MAC_ADDRESS_3" : UInt = PLC WP231PR_DB.DR12.DEVICE_MAC_ADDRESS_3 AT %DB231.DBW1060, 1 s
   "WP231PR_DB_DR12_DEVICE_MAC_ADDRESS_4" : UInt = PLC WP231PR_DB.DR12.DEVICE_MAC_ADDRESS_4 AT %DB231.DBW1062, 1 s
   "WP231PR_DB_DR12_DEVICE_MAC_ADDRESS_5" : UInt = PLC WP231PR_DB.DR12.DEVICE_MAC_ADDRESS_5 AT %DB231.DBW1064, 1 s
   "WP231PR_DB_DR12_PORT_MAC_ADDRESS" : UInt = PLC WP231PR_DB.DR12.PORT_MAC_ADDRESS AT %DB231.DBW1066, 1 s
   "WP231PR_DB_DR12_PORT_MAC_ADDRESS_1" : UInt = PLC WP231PR_DB.DR12.PORT_MAC_ADDRESS_1 AT %DB231.DBW1068, 1 s
   "WP231PR_DB_DR12_PORT_MAC_ADDRESS_2" : UInt = PLC WP231PR_DB.DR12.PORT_MAC_ADDRESS_2 AT %DB231.DBW1070, 1 s
   "WP231PR_DB_DR12_PORT_MAC_ADDRESS_3" : UInt = PLC WP231PR_DB.DR12.PORT_MAC_ADDRESS_3 AT %DB231.DBW1072, 1 s
   "WP231PR_DB_DR12_PORT_MAC_ADDRESS_4" : UInt = PLC WP231PR_DB.DR12.PORT_MAC_ADDRESS_4 AT %DB231.DBW1074, 1 s
   "WP231PR_DB_DR12_PORT_MAC_ADDRESS_5" : UInt = PLC WP231PR_DB.DR12.PORT_MAC_ADDRESS_5 AT %DB231.DBW1076, 1 s
   "WP231PR_DB_DR12_IP_ADDRESS_1" : UInt = PLC WP231PR_DB.DR12.IP_ADDRESS_1 AT %DB231.DBW1078, 1 s
   "WP231PR_DB_DR12_IP_ADDRESS_2" : UInt = PLC WP231PR_DB.DR12.IP_ADDRESS_2 AT %DB231.DBW1080, 1 s
   "WP231PR_DB_DR12_IP_ADDRESS_3" : UInt = PLC WP231PR_DB.DR12.IP_ADDRESS_3 AT %DB231.DBW1082, 1 s
   "WP231PR_DB_DR12_IP_ADDRESS_4" : UInt = PLC WP231PR_DB.DR12.IP_ADDRESS_4 AT %DB231.DBW1084, 1 s
   "WP231PR_DB_DR12_SUB_NET_MASK_1" : UInt = PLC WP231PR_DB.DR12.SUB_NET_MASK_1 AT %DB231.DBW1086, 1 s
   "WP231PR_DB_DR12_SUB_NET_MASK_2" : UInt = PLC WP231PR_DB.DR12.SUB_NET_MASK_2 AT %DB231.DBW1088, 1 s
   "WP231PR_DB_DR12_SUB_NET_MASK_3" : UInt = PLC WP231PR_DB.DR12.SUB_NET_MASK_3 AT %DB231.DBW1090, 1 s
   "WP231PR_DB_DR12_SUB_NET_MASK_4" : UInt = PLC WP231PR_DB.DR12.SUB_NET_MASK_4 AT %DB231.DBW1092, 1 s
   "WP231PR_DB_DR12_CURRENT_GATEWAY_1" : UInt = PLC WP231PR_DB.DR12.CURRENT_GATEWAY_1 AT %DB231.DBW1094, 1 s
   "WP231PR_DB_DR12_CURRENT_GATEWAY_2" : UInt = PLC WP231PR_DB.DR12.CURRENT_GATEWAY_2 AT %DB231.DBW1096, 1 s
   "WP231PR_DB_DR12_CURRENT_GATEWAY_3" : UInt = PLC WP231PR_DB.DR12.CURRENT_GATEWAY_3 AT %DB231.DBW1098, 1 s
   "WP231PR_DB_DR12_CURRENT_GATEWAY_4" : UInt = PLC WP231PR_DB.DR12.CURRENT_GATEWAY_4 AT %DB231.DBW1100, 1 s

HMI tags "Data Record DR13"
   "WP231PR_DB_DR13_RS485_PROTOCOL" : UInt = PLC WP231PR_DB.DR13.RS485_PROTOCOL AT %DB231.DBW1154, 1 s
   "WP231PR_DB_DR13_RS485_BAUD_RATE" : UInt = PLC WP231PR_DB.DR13.RS485_BAUD_RATE AT %DB231.DBW1156, 1 s
   "WP231PR_DB_DR13_RS485_PARITY" : Bool = PLC WP231PR_DB.DR13.RS485_PARITY AT %DB231.DBX1159.0, 1 s
   "WP231PR_DB_DR13_RS485_DATA_BITS" : Bool = PLC WP231PR_DB.DR13.RS485_DATA_BITS AT %DB231.DBX1159.1, 1 s
   "WP231PR_DB_DR13_RS485_STOP_BITS" : Bool = PLC WP231PR_DB.DR13.RS485_STOP_BITS AT %DB231.DBX1159.2, 1 s
   "WP231PR_DB_DR13_MODBUS_RTU_ADDRESS" : UInt = PLC WP231PR_DB.DR13.MODBUS_RTU_ADDRESS AT %DB231.DBW1160, 1 s
   "WP231PR_DB_DR13_DEC_POINT_REM_DISPLAY" : Int = PLC WP231PR_DB.DR13.DEC_POINT_REM_DISPLAY AT %DB231.DBW1162, 1 s
   "WP231PR_DB_DR13_MODBUS_RTU_RESPONSE_DELAY" : UInt = PLC WP231PR_DB.DR13.MODBUS_RTU_RESPONSE_DELAY AT %DB231.DBW1164, 1 s

HMI tags "Data Record DR14"
   "WP231PR_DB_DR14_SEL_PROC_VAL_1_SIMATIC" : UInt = PLC WP231PR_DB.DR14.SEL_PROC_VAL_1_SIMATIC AT %DB231.DBW1178, 1 s
   "WP231PR_DB_DR14_SEL_PROC_VAL_2_SIMATIC" : UInt = PLC WP231PR_DB.DR14.SEL_PROC_VAL_2_SIMATIC AT %DB231.DBW1180, 1 s

HMI tags "Data Record DR15"
   "WP231PR_DB_DR15_PRESET_TARE_1" : Real = PLC WP231PR_DB.DR15.PRESET_TARE_1 AT %DB231.DBD1194, 1 s
   "WP231PR_DB_DR15_PRESET_TARE_2" : Real = PLC WP231PR_DB.DR15.PRESET_TARE_2 AT %DB231.DBD1198, 1 s
   "WP231PR_DB_DR15_PRESET_TARE_3" : Real = PLC WP231PR_DB.DR15.PRESET_TARE_3 AT %DB231.DBD1202, 1 s

HMI tags "Data Record DR16"
   "WP231PR_DB_DR16_SIMULATION_WEIGHT" : Real = PLC WP231PR_DB.DR16.SIMULATION_WEIGHT AT %DB231.DBD1222, 1 s

HMI tags "Data Record DR17"
   "WP231PR_DB_DR17_ANA_OUT_VALUE" : Real = PLC WP231PR_DB.DR17.ANA_OUT_VALUE AT %DB231.DBD1238, 1 s

HMI tags "Data Record DR18"
   "WP231PR_DB_DR18_DEF_DIG_OUT_DQ_0" : Bool = PLC WP231PR_DB.DR18.DEF_DIG_OUT_DQ_0 AT %DB231.DBX1255.0, 1 s
   "WP231PR_DB_DR18_DEF_DIG_OUT_DQ_1" : Bool = PLC WP231PR_DB.DR18.DEF_DIG_OUT_DQ_1 AT %DB231.DBX1255.1, 1 s
   "WP231PR_DB_DR18_DEF_DIG_OUT_DQ_2" : Bool = PLC WP231PR_DB.DR18.DEF_DIG_OUT_DQ_2 AT %DB231.DBX1255.2, 1 s
   "WP231PR_DB_DR18_DEF_DIG_OUT_DQ_3" : Bool = PLC WP231PR_DB.DR18.DEF_DIG_OUT_DQ_3 AT %DB231.DBX1255.3, 1 s

HMI tags "Data Record DR30"
   "WP231PR_DB_DR30_OPERATION_ERRORS" : UInt = PLC WP231PR_DB.DR30.OPERATION_ERRORS AT %DB231.DBW1270, 1 s
   "WP231PR_DB_DR30_TECHNOLOGICAL_ERRORS" : UInt = PLC WP231PR_DB.DR30.TECHNOLOGICAL_ERRORS AT %DB231.DBW1272, 1 s
   "WP231PR_DB_DR30_GROSS_PROCESS" : Real = PLC WP231PR_DB.DR30.GROSS_PROCESS AT %DB231.DBD1274, 500 ms
   "WP231PR_DB_DR30_NET_PROCESS" : Real = PLC WP231PR_DB.DR30.NET_PROCESS AT %DB231.DBD1278, 1 s
   "WP231PR_DB_DR30_TARE_PROCESS" : Real = PLC WP231PR_DB.DR30.TARE_PROCESS AT %DB231.DBD1282, 1 s
   "WP231PR_DB_DR30_GROSS_NET_WEIGHT" : Real = PLC WP231PR_DB.DR30.GROSS_NET_WEIGHT AT %DB231.DBD1286, 1 s
   "WP231PR_DB_DR30_GROSS_NET_WEIGHT_X10" : Real = PLC WP231PR_DB.DR30.GROSS_NET_WEIGHT_X10 AT %DB231.DBD1290, 1 s
   "WP231PR_DB_DR30_TARE" : Real = PLC WP231PR_DB.DR30.TARE AT %DB231.DBD1294, 1 s
   "WP231PR_DB_DR30_GROSS_PROCESS_2" : Real = PLC WP231PR_DB.DR30.GROSS_PROCESS_2 AT %DB231.DBD1298, 1 s
   "WP231PR_DB_DR30_NET_PROCESS_2" : Real = PLC WP231PR_DB.DR30.NET_PROCESS_2 AT %DB231.DBD1302, 1 s
   "WP231PR_DB_DR30_REFRESH_COUNTER" : UInt = PLC WP231PR_DB.DR30.REFRESH_COUNTER AT %DB231.DBW1306, 1 s
   "WP231PR_DB_DR30_LAST_PROTOCOL_ID" : UDInt = PLC WP231PR_DB.DR30.LAST_PROTOCOL_ID AT %DB231.DBD1310, 1 s

HMI tags "Data Record DR31"
   "WP231PR_DB_DR31_DIGITS_UNFILTERED" : DInt = PLC WP231PR_DB.DR31.DIGITS_UNFILTERED AT %DB231.DBD1326, 1 s
   "WP231PR_DB_DR31_DIGITS_FILTERED" : DInt = PLC WP231PR_DB.DR31.DIGITS_FILTERED AT %DB231.DBD1330, 1 s
   "WP231PR_DB_DR31_DIGITS_2_FILTERED" : DInt = PLC WP231PR_DB.DR31.DIGITS_2_FILTERED AT %DB231.DBD1334, 1 s
   "WP231PR_DB_DR31_CURRENT_ANA_OUT_DIGITS" : UInt = PLC WP231PR_DB.DR31.CURRENT_ANA_OUT_DIGITS AT %DB231.DBW1340, 1 s
   "WP231PR_DB_DR31_CURRENT_STATE_DQ_0" : Bool = PLC WP231PR_DB.DR31.CURRENT_STATE_DQ_0 AT %DB231.DBX1342.0, 1 s
   "WP231PR_DB_DR31_CURRENT_STATE_DQ_1" : Bool = PLC WP231PR_DB.DR31.CURRENT_STATE_DQ_1 AT %DB231.DBX1342.1, 1 s
   "WP231PR_DB_DR31_CURRENT_STATE_DQ_2" : Bool = PLC WP231PR_DB.DR31.CURRENT_STATE_DQ_2 AT %DB231.DBX1342.2, 1 s
   "WP231PR_DB_DR31_CURRENT_STATE_DQ_3" : Bool = PLC WP231PR_DB.DR31.CURRENT_STATE_DQ_3 AT %DB231.DBX1342.3, 1 s
   "WP231PR_DB_DR31_CURRENT_STATE_DI_0" : Bool = PLC WP231PR_DB.DR31.CURRENT_STATE_DI_0 AT %DB231.DBX1343.0, 1 s
   "WP231PR_DB_DR31_CURRENT_STATE_DI_1" : Bool = PLC WP231PR_DB.DR31.CURRENT_STATE_DI_1 AT %DB231.DBX1343.1, 1 s
   "WP231PR_DB_DR31_CURRENT_STATE_DI_2" : Bool = PLC WP231PR_DB.DR31.CURRENT_STATE_DI_2 AT %DB231.DBX1343.2, 1 s
   "WP231PR_DB_DR31_CURRENT_STATE_DI_3" : Bool = PLC WP231PR_DB.DR31.CURRENT_STATE_DI_3 AT %DB231.DBX1343.3, 1 s
   "WP231PR_DB_DR31_DIP_SWITCH_1" : Bool = PLC WP231PR_DB.DR31.DIP_SWITCH_1 AT %DB231.DBX1343.6, 1 s
   "WP231PR_DB_DR31_DIP_SWITCH_2" : Bool = PLC WP231PR_DB.DR31.DIP_SWITCH_2 AT %DB231.DBX1343.7, 1 s
   "WP231PR_DB_DR31_REFRESH_COUNTER" : UInt = PLC WP231PR_DB.DR31.REFRESH_COUNTER AT %DB231.DBW1344, 1 s
   "WP231PR_DB_DR31_LOAD_CELL_SIGNAL" : Real = PLC WP231PR_DB.DR31.LOAD_CELL_SIGNAL AT %DB231.DBD1346, 1 s

HMI tags "Data Record DR32"
   "WP231PR_DB_DR32_DATA_CMD_ERR_1" : UInt = PLC WP231PR_DB.DR32.DATA_CMD_ERR_1 AT %DB231.DBW1358, 1 s
   "WP231PR_DB_DR32_DATA_CMD_ERR_2" : UInt = PLC WP231PR_DB.DR32.DATA_CMD_ERR_2 AT %DB231.DBW1360, 1 s
   "WP231PR_DB_DR32_DATA_CMD_ERR_3" : UInt = PLC WP231PR_DB.DR32.DATA_CMD_ERR_3 AT %DB231.DBW1362, 1 s
   "WP231PR_DB_DR32_DATA_CMD_ERR_4" : UInt = PLC WP231PR_DB.DR32.DATA_CMD_ERR_4 AT %DB231.DBW1364, 1 s
   "WP231PR_DB_DR32_ERR_CODE_S7_INTERFACE" : UInt = PLC WP231PR_DB.DR32.ERR_CODE_S7_INTERFACE AT %DB231.DBW1366, 1 s
   "WP231PR_DB_DR32_ERR_CODE_MODBUS_RS485" : UInt = PLC WP231PR_DB.DR32.ERR_CODE_MODBUS_RS485 AT %DB231.DBW1368, 1 s
   "WP231PR_DB_DR32_ERR_CODE_MODBUS_ETH" : UInt = PLC WP231PR_DB.DR32.ERR_CODE_MODBUS_ETH AT %DB231.DBW1370, 1 s
   "WP231PR_DB_DR32_ERR_CODE_SIWATOOL" : UInt = PLC WP231PR_DB.DR32.ERR_CODE_SIWATOOL AT %DB231.DBW1372, 1 s
   "WP231PR_DB_DR32_CMD_ERR_DI" : UInt = PLC WP231PR_DB.DR32.CMD_ERR_DI AT %DB231.DBW1374, 1 s

HMI tags "Data Record DR34"
   "WP231PR_DB_DR34_ASCII_DISPLAY" : String[16] = PLC WP231PR_DB.DR34.ASCII_DISPLAY AT %DB231.DBX1386.0, 100 ms

HMI tags "Data Record DR45"
   "WP231PR_DB_DR45_PROTOCOL_ID_TO_READ" : String[12] = PLC WP231PR_DB.DR45.PROTOCOL_ID_TO_READ AT %DB231.DBX1596.0, 1 s
   "WP231PR_DB_DR45_PROTOCOL_ID_TO_READ_DEC" : DInt = PLC WP231PR_DB.DR45.PROTOCOL_ID_TO_READ_DEC AT %DB231.DBD1612, 1 s

HMI tags "Data Record DR46"
   "WP231PR_DB_DR46_OLDEST_LOG_ID_DEC" : UDInt = PLC WP231PR_DB.DR46.OLDEST_LOG_ID_DEC AT %DB231.DBD1624, 1 s
   "WP231PR_DB_DR46_LAST_LOG_ID_DEC" : UDInt = PLC WP231PR_DB.DR46.LAST_LOG_ID_DEC AT %DB231.DBD1628, 1 s
   "WP231PR_DB_DR46_SELECTED_PROTOCOL_ID_DEC" : UDInt = PLC WP231PR_DB.DR46.SELECTED_PROTOCOL_ID_DEC AT %DB231.DBD1632, 1 s
   "WP231PR_DB_DR46_OLDEST_LOG_ID" : String[12] = PLC WP231PR_DB.DR46.OLDEST_LOG_ID AT %DB231.DBX1636.0, 1 s
   "WP231PR_DB_DR46_LAST_LOG_ID" : String[12] = PLC WP231PR_DB.DR46.LAST_LOG_ID AT %DB231.DBX1650.0, 1 s
   "WP231PR_DB_DR46_SELECTED_PROTOCOL_ID" : String[12] = PLC WP231PR_DB.DR46.SELECTED_PROTOCOL_ID AT %DB231.DBX1664.0, 1 s
   "WP231PR_DB_DR46_PROTOCOL_STRING" : String[28] = PLC WP231PR_DB.DR46.PROTOCOL_STRING AT %DB231.DBX1678.0, 1 s
   "WP231PR_DB_DR46_CHECKSUM" : String[4] = PLC WP231PR_DB.DR46.CHECKSUM AT %DB231.DBX1708.0, 1 s
   "WP231PR_DB_DR46_PROTOCOL_DATE" : String[10] = PLC WP231PR_DB.DR46.PROTOCOL_DATE AT %DB231.DBX1714.0, 1 s
   "WP231PR_DB_DR46_PROTOCOL_TIME" : String[8] = PLC WP231PR_DB.DR46.PROTOCOL_TIME AT %DB231.DBX1726.0, 1 s
   "WP231PR_DB_DR46_ADD_INFORMATION" : String[4] = PLC WP231PR_DB.DR46.ADD_INFORMATION AT %DB231.DBX1736.0, 1 s

HMI tags "Data Record DR47"
   "WP231PR_DB_DR47_OLDEST_LOG_ID" : String[8] = PLC WP231PR_DB.DR47.OLDEST_LOG_ID AT %DB231.DBX1752.0, 1 s
   "WP231PR_DB_DR47_LAST_LOG_ID" : String[8] = PLC WP231PR_DB.DR47.LAST_LOG_ID AT %DB231.DBX1762.0, 1 s
   "WP231PR_DB_DR47_SELECTED_LOG" : String[8] = PLC WP231PR_DB.DR47.SELECTED_LOG AT %DB231.DBX1772.0, 1 s
   "WP231PR_DB_DR47_DEVICE" : String[4] = PLC WP231PR_DB.DR47.DEVICE AT %DB231.DBX1782.0, 1 s
   "WP231PR_DB_DR47_FW_VERSION_OLD" : String[10] = PLC WP231PR_DB.DR47.FW_VERSION_OLD AT %DB231.DBX1788.0, 1 s
   "WP231PR_DB_DR47_FW_VERSION_NEW" : String[10] = PLC WP231PR_DB.DR47.FW_VERSION_NEW AT %DB231.DBX1800.0, 1 s
   "WP231PR_DB_DR47_CHECKSUM" : UInt = PLC WP231PR_DB.DR47.CHECKSUM AT %DB231.DBW1812, 1 s

HMI tags "Data Record DR48"
   "WP231PR_DB_DR48_YEAR" : UInt = PLC WP231PR_DB.DR48.YEAR AT %DB231.DBW1824, 1 s
   "WP231PR_DB_DR48_MONTH" : UInt = PLC WP231PR_DB.DR48.MONTH AT %DB231.DBW1826, 1 s
   "WP231PR_DB_DR48_DAY" : UInt = PLC WP231PR_DB.DR48.DAY AT %DB231.DBW1828, 1 s
   "WP231PR_DB_DR48_HOUR" : UInt = PLC WP231PR_DB.DR48.HOUR AT %DB231.DBW1830, 1 s
   "WP231PR_DB_DR48_MINUTE" : UInt = PLC WP231PR_DB.DR48.MINUTE AT %DB231.DBW1832, 1 s
   "WP231PR_DB_DR48_SECOND" : UInt = PLC WP231PR_DB.DR48.SECOND AT %DB231.DBW1834, 1 s
   "WP231PR_DB_DR48_MSECOND" : UInt = PLC WP231PR_DB.DR48.MSECOND AT %DB231.DBW1836, 1 s
   "WP231PR_DB_DR48_DAY_OF_WEEK" : UInt = PLC WP231PR_DB.DR48.DAY_OF_WEEK AT %DB231.DBW1838, 1 s

HMI tags "CMD"
   "WP231PR_DB_s_CMD1_i_CMD_CODE" : Int = PLC WP231PR_DB.s_CMD1.i_CMD_CODE AT %DB231.DBW462, 1 s
   "WP231PR_DB_s_CMD1_bo_CMD_TRIGGER" : Bool = PLC WP231PR_DB.s_CMD1.bo_CMD_TRIGGER AT %DB231.DBX464.0, 1 s
   "WP231PR_DB_s_CMD2_i_CMD_CODE" : Int = PLC WP231PR_DB.s_CMD2.i_CMD_CODE AT %DB231.DBW466, 1 s
   "WP231PR_DB_s_CMD2_bo_CMD_TRIGGER" : Bool = PLC WP231PR_DB.s_CMD2.bo_CMD_TRIGGER AT %DB231.DBX468.0, 1 s
   "WP231PR_DB_s_CMD3_i_CMD_CODE" : Int = PLC WP231PR_DB.s_CMD3.i_CMD_CODE AT %DB231.DBW470, 1 s
   "WP231PR_DB_s_CMD3_bo_CMD_TRIGGER" : Bool = PLC WP231PR_DB.s_CMD3.bo_CMD_TRIGGER AT %DB231.DBX472.0, 1 s
   "WP231PR_DB_CMD_A" : Int = PLC WP231PR_DB.CMD_A AT %DB231.DBW458, 1 s
   "WP231PR_DB_CMD_B" : Int = PLC WP231PR_DB.CMD_B AT %DB231.DBW460, 1 s

HMI tags "IO_Data"
   "WP231PR_DB_s_IO_DATA_OPERATION_ERRORS" : UInt = PLC WP231PR_DB.s_IO_DATA.OPERATION_ERRORS AT %DB231.DBW508, 100 ms
   "WP231PR_DB_s_IO_DATA_TECHNOLOGICAL_ERRORS" : UInt = PLC WP231PR_DB.s_IO_DATA.TECHNOLOGICAL_ERRORS AT %DB231.DBW510, 100 ms
   "WP231PR_DB_s_IO_DATA_DATA_CMD_ERROR_1" : UInt = PLC WP231PR_DB.s_IO_DATA.DATA_CMD_ERROR_1 AT %DB231.DBW512, 100 ms
   "WP231PR_DB_s_IO_DATA_DATA_CMD_ERROR_2" : UInt = PLC WP231PR_DB.s_IO_DATA.DATA_CMD_ERROR_2 AT %DB231.DBW514, 100 ms
   "WP231PR_DB_s_IO_DATA_DATA_CMD_ERROR_3" : UInt = PLC WP231PR_DB.s_IO_DATA.DATA_CMD_ERROR_3 AT %DB231.DBW516, 100 ms
   "WP231PR_DB_s_IO_DATA_DATA_CMD_ERROR_4" : UInt = PLC WP231PR_DB.s_IO_DATA.DATA_CMD_ERROR_4 AT %DB231.DBW518, 100 ms
   "WP231PR_DB_s_IO_DATA_SCALE_STATUS_1_EMPTY" : Bool = PLC WP231PR_DB.s_IO_DATA.SCALE_STATUS_1.EMPTY AT %DB231.DBX488.0, 100 ms
   "WP231PR_DB_s_IO_DATA_SCALE_STATUS_1_LIMIT_1" : Bool = PLC WP231PR_DB.s_IO_DATA.SCALE_STATUS_1.LIMIT_1 AT %DB231.DBX488.1, 100 ms
   "WP231PR_DB_s_IO_DATA_SCALE_STATUS_1_LIMIT_2" : Bool = PLC WP231PR_DB.s_IO_DATA.SCALE_STATUS_1.LIMIT_2 AT %DB231.DBX488.2, 100 ms
   "WP231PR_DB_s_IO_DATA_SCALE_STATUS_1_BELOW_MIN_WEIGHT" : Bool = PLC WP231PR_DB.s_IO_DATA.SCALE_STATUS_1.BELOW_MIN_WEIGHT AT %DB231.DBX488.3, 100 ms
   "WP231PR_DB_s_IO_DATA_SCALE_STATUS_1_D_ZERO" : Bool = PLC WP231PR_DB.s_IO_DATA.SCALE_STATUS_1.D_ZERO AT %DB231.DBX489.0, 100 ms
   "WP231PR_DB_s_IO_DATA_SCALE_STATUS_1_MAX_9E" : Bool = PLC WP231PR_DB.s_IO_DATA.SCALE_STATUS_1.MAX_9E AT %DB231.DBX489.1, 100 ms
   "WP231PR_DB_s_IO_DATA_SCALE_STATUS_1_TARE" : Bool = PLC WP231PR_DB.s_IO_DATA.SCALE_STATUS_1.TARE AT %DB231.DBX489.2, 100 ms
   "WP231PR_DB_s_IO_DATA_SCALE_STATUS_1_PRESET_TARE" : Bool = PLC WP231PR_DB.s_IO_DATA.SCALE_STATUS_1.PRESET_TARE AT %DB231.DBX489.3, 100 ms
   "WP231PR_DB_s_IO_DATA_SCALE_STATUS_1_WAITING_FOR_STANDSTILL" : Bool = PLC WP231PR_DB.s_IO_DATA.SCALE_STATUS_1.WAITING_FOR_STANDSTILL AT %DB231.DBX489.5, 100 ms
   "WP231PR_DB_s_IO_DATA_SCALE_STATUS_1_STANDSTILL" : Bool = PLC WP231PR_DB.s_IO_DATA.SCALE_STATUS_1.STANDSTILL AT %DB231.DBX489.6, 100 ms
   "WP231PR_DB_s_IO_DATA_SCALE_STATUS_2_CALIBRATED" : Bool = PLC WP231PR_DB.s_IO_DATA.SCALE_STATUS_2.CALIBRATED AT %DB231.DBX490.0, 100 ms
   "WP231PR_DB_s_IO_DATA_SCALE_STATUS_2_SERVICE_MODE" : Bool = PLC WP231PR_DB.s_IO_DATA.SCALE_STATUS_2.SERVICE_MODE AT %DB231.DBX490.1, 100 ms
   "WP231PR_DB_s_IO_DATA_SCALE_STATUS_2_SIMULATION_MODE" : Bool = PLC WP231PR_DB.s_IO_DATA.SCALE_STATUS_2.SIMULATION_MODE AT %DB231.DBX490.2, 100 ms
   "WP231PR_DB_s_IO_DATA_SCALE_STATUS_2_WRITE_PROTECTION" : Bool = PLC WP231PR_DB.s_IO_DATA.SCALE_STATUS_2.WRITE_PROTECTION AT %DB231.DBX490.3, 100 ms
   "WP231PR_DB_s_IO_DATA_SCALE_STATUS_2_ANALOGUE_OUT_ERROR" : Bool = PLC WP231PR_DB.s_IO_DATA.SCALE_STATUS_2.ANALOGUE_OUT_ERROR AT %DB231.DBX490.4, 100 ms
   "WP231PR_DB_s_IO_DATA_SCALE_STATUS_2_START_UP" : Bool = PLC WP231PR_DB.s_IO_DATA.SCALE_STATUS_2.START_UP AT %DB231.DBX490.6, 100 ms
   "WP231PR_DB_s_IO_DATA_SCALE_STATUS_2_ERROR" : Bool = PLC WP231PR_DB.s_IO_DATA.SCALE_STATUS_2.ERROR AT %DB231.DBX490.7, 100 ms
   "WP231PR_DB_s_IO_DATA_SCALE_STATUS_2_TIME_BUFFER_ERROR" : Bool = PLC WP231PR_DB.s_IO_DATA.SCALE_STATUS_2.TIME_BUFFER_ERROR AT %DB231.DBX491.5, 100 ms
   "WP231PR_DB_s_IO_DATA_SCALE_STATUS_2_TRACE" : Bool = PLC WP231PR_DB.s_IO_DATA.SCALE_STATUS_2.TRACE AT %DB231.DBX491.6, 100 ms
   "WP231PR_DB_s_IO_DATA_SCALE_STATUS_2_DIGITAL_INPUT_ERROR" : Bool = PLC WP231PR_DB.s_IO_DATA.SCALE_STATUS_2.DIGITAL_INPUT_ERROR AT %DB231.DBX491.7, 100 ms

HMI tags "INTERNAL"
   "S1_DISPLAY_TAG" : Bool, internal
   "S1_LOADCURVE_MIN" : Real, internal
   "S1_SHOW_HELP" : Bool, internal
   "SecureDisplayRunning" : Bool AT %DB1.DBX0.0

discrete alarms
   7: 'В системе нет коробок', class Errors, trigger "Logic_DB_Alarm" bit 0
   8: 'Т 0 - Выбило защитный автомат', class Errors, trigger "Motors_DB_T0_Alarm" bit 0
   9: 'Т 0 - Ошибка при запуске', class Errors, trigger "Motors_DB_T0_Alarm" bit 1
   10: 'Т 0 - Ошибка при останове', class Errors, trigger "Motors_DB_T0_Alarm" bit 2
   11: 'Т 0 - Сработало реле безопасности', class Errors, trigger "Motors_DB_T0_Alarm" bit 3
   12: 'Т 0 - Общая блокировка', class Errors, trigger "Motors_DB_T0_Alarm" bit 4
   13: 'Т 0 - Перегрев двигателя', class Errors, trigger "Motors_DB_T0_Alarm" bit 5
   14: 'Т 1 - Выбило защитный автомат', class Errors, trigger "Motors_DB_T1_Alarm" bit 0
   15: 'Т 1 - Ошибка при запуске', class Errors, trigger "Motors_DB_T1_Alarm" bit 1
   16: 'Т 1 - Ошибка при останове', class Errors, trigger "Motors_DB_T1_Alarm" bit 2
   17: 'Т 1 - Сработало реле безопасности', class Errors, trigger "Motors_DB_T1_Alarm" bit 3
   18: 'Т 1 - Общая блокировка', class Errors, trigger "Motors_DB_T1_Alarm" bit 4
   19: 'Т 1 - Перегрев двигателя', class Errors, trigger "Motors_DB_T1_Alarm" bit 5
   20: 'Т 2 - Выбило защитный автомат', class Errors, trigger "Motors_DB_T2_Alarm" bit 0
   21: 'Т 2 - Ошибка при запуске', class Errors, trigger "Motors_DB_T2_Alarm" bit 1
   22: 'Т 2 - Ошибка при останове', class Errors, trigger "Motors_DB_T2_Alarm" bit 2
   23: 'Т 2 - Сработало реле безопасности', class Errors, trigger "Motors_DB_T2_Alarm" bit 3
   24: 'Т 2 - Общая блокировка', class Errors, trigger "Motors_DB_T2_Alarm" bit 4
   25: 'Т 2 - Перегрев двигателя', class Errors, trigger "Motors_DB_T2_Alarm" bit 5
   26: 'Т 3 - Выбило защитный автомат', class Errors, trigger "Motors_DB_T3_Alarm" bit 0
   27: 'Т 3 - Ошибка при запуске', class Errors, trigger "Motors_DB_T3_Alarm" bit 1
   28: 'Т 3 - Ошибка при останове', class Errors, trigger "Motors_DB_T3_Alarm" bit 2
   29: 'Т 3 - Сработало реле безопасности', class Errors, trigger "Motors_DB_T3_Alarm" bit 3
   30: 'Т 3 - Общая блокировка', class Errors, trigger "Motors_DB_T3_Alarm" bit 4
   31: 'Т 3 - Перегрев двигателя', class Errors, trigger "Motors_DB_T3_Alarm" bit 5
   32: 'Т 4 - Выбило защитный автомат', class Errors, trigger "Motors_DB_T4_Alarm" bit 0
   33: 'Т 4 - Ошибка при запуске', class Errors, trigger "Motors_DB_T4_Alarm" bit 1
   34: 'Т 4 - Ошибка при останове', class Errors, trigger "Motors_DB_T4_Alarm" bit 2
   35: 'Т 4 - Сработало реле безопасности', class Errors, trigger "Motors_DB_T4_Alarm" bit 3
   36: 'Т 4 - Общая блокировка', class Errors, trigger "Motors_DB_T4_Alarm" bit 4
   37: 'Т 4 - Перегрев двигателя', class Errors, trigger "Motors_DB_T4_Alarm" bit 5
   38: 'V 1 - Выбило защитный автомат', class Errors, trigger "Valves_DB_V1_Alarm" bit 0
   39: 'V 1 - Не сработал пускатель - открыто', class Errors, trigger "Valves_DB_V1_Alarm" bit 1
   40: 'V 1 - Не сработал пускатель - закрыто', class Errors, trigger "Valves_DB_V1_Alarm" bit 2
   41: 'V 1 - Не сработал концевик - открыто', class Errors, trigger "Valves_DB_V1_Alarm" bit 3
   42: 'V 1 - Не сработал концевик - закрыто', class Errors, trigger "Valves_DB_V1_Alarm" bit 4
   43: 'V 1 - Две ОС', class Errors, trigger "Valves_DB_V1_Alarm" bit 5
   44: 'V 1 - Аварийная остановка', class Errors, trigger "Valves_DB_V1_Alarm" bit 6
   45: 'V 2 - Выбило защитный автомат', class Errors, trigger "Valves_DB_V2_Alarm" bit 0
   46: 'V 2 - Не сработал пускатель - открыто', class Errors, trigger "Valves_DB_V2_Alarm" bit 1
   47: 'V 2 - Не сработал пускатель - закрыто', class Errors, trigger "Valves_DB_V2_Alarm" bit 2
   48: 'V 2 - Не сработал концевик - открыто', class Errors, trigger "Valves_DB_V2_Alarm" bit 3
   49: 'V 2 - Не сработал концевик - закрыто', class Errors, trigger "Valves_DB_V2_Alarm" bit 4
   50: 'V 2 - Две ОС', class Errors, trigger "Valves_DB_V2_Alarm" bit 5
   51: 'V 2 - Аварийная остановка', class Errors, trigger "Valves_DB_V2_Alarm" bit 6
   52: 'V 3 - Выбило защитный автомат', class Errors, trigger "Valves_DB_V3_Alarm" bit 0
   53: 'V 3 - Не сработал пускатель - открыто', class Errors, trigger "Valves_DB_V3_Alarm" bit 1
   54: 'V 3 - Не сработал пускатель - закрыто', class Errors, trigger "Valves_DB_V3_Alarm" bit 2
   55: 'V 3 - Не сработал концевик - открыто', class Errors, trigger "Valves_DB_V3_Alarm" bit 3
   56: 'V 3 - Не сработал концевик - закрыто', class Errors, trigger "Valves_DB_V3_Alarm" bit 4
   57: 'V 3 - Две ОС', class Errors, trigger "Valves_DB_V3_Alarm" bit 5
   58: 'V 3 - Аварийная остановка', class Errors, trigger "Valves_DB_V3_Alarm" bit 6
   59: 'Статистика - Переполнение памяти', class Errors, trigger "T3V3W3_DB_Alarm" bit 0
   60: 'Статистика - Переполнение колличества партий', class Errors, trigger "T3V3W3_DB_Alarm" bit 1
   1: 'Статистика - Ошибка записи файла', class Errors, trigger "del_stat_mem_DB_Alarm" bit 0
   2: 'Статистика - Партия в процессе записи', class Errors, trigger "del_stat_mem_DB_Alarm" bit 1
   3: 'Статистика - Имя уже используется', class Errors, trigger "T3V3W3_DB_Alarm" bit 2
   4: 'Статистика - Недопустимое имя', class Errors, trigger "T3V3W3_DB_Alarm" bit 3
   97: '1006 Fehler Logbuch / 1006 Error log-book / 1006 Erreur sur le cahier des rapports', class Errors, trigger "WP231PR_DB_s_IO_DATA_OPERATION_ERRORS" bit 12
   98: '5000 Daten- oder Bedienfehler / 5000 Data or command error / 5000 Erreur données ou utilisateur', class Errors, trigger "WP231PR_DB_s_IO_DATA_DATA_CMD_ERROR_1" bit 0
   99: '5001 Befehlscode oder Datensatz nicht bekannt / 5001 Data record or command unknown / 5001 Ordre ou numéro de DR inconnu', class Errors, trigger "WP231PR_DB_s_IO_DATA_DATA_CMD_ERROR_1" bit 1
   100: '5002 Befehl oder Datenänderung nicht erlaubt, da Schreibschutz aktiv / 5002 Command or Data modification not allowed / 5002 Ordre ou modification des paramètres interdit parce que la protection en écriture est activée', class Errors, trigger "WP231PR_DB_s_IO_DATA_DATA_CMD_ERROR_1" bit 2
   101: '5003 Verlassen des Servicebetriebs unzulässig, da Justage nicht abgeschlossen / 5003 Service Mode can't be switched off, as calibration was not completed / 5003 Impossible de quitter le mode service parce que l'étalonnage n'est pas terminé', class Errors, trigger "WP231PR_DB_s_IO_DATA_DATA_CMD_ERROR_1" bit 3
   102: '5004 Befehl oder Datenübertragung nur im Servicebetrieb möglich / 5004 Command or data transfer only permitted in service mode / 5004 Ordre ou transmission de données uniquement possible en mode service', class Errors, trigger "WP231PR_DB_s_IO_DATA_DATA_CMD_ERROR_1" bit 4
   103: '5005 Befehl oder Datenübertragung im Servicebetrieb nicht möglich, da Servicebetrieb aktiv / 5005 Command or data transfer not permitted in service mode / 5005 Ordre ou transmission de données impossible parce que le mode service est activé', class Errors, trigger "WP231PR_DB_s_IO_DATA_DATA_CMD_ERROR_1" bit 5
   104: '5006 Befehl oder Datenübertragung nicht möglich da BUSY / 5006 Command or data transfer not possible while BUSY / 5006 Ordre ou transmission de données impossible parce que la CPU est en mode stop ou erreur', class Errors, trigger "WP231PR_DB_s_IO_DATA_DATA_CMD_ERROR_1" bit 6
   105: '5007 Befehl oder Datenübertragung nicht möglich da Modul gestört oder CPU in Stop / 5007 Command or data transfer not possible because of error or CPU stop / 5007 Ordre ou transmission de données impossible parce que le module est en mode BUSY', class Errors, trigger "WP231PR_DB_s_IO_DATA_DATA_CMD_ERROR_1" bit 7
   106: 'Daten-Bedienfehler Byte 2 Bit 0 / Data Command Error Byte 2 Bit 0 / Erreur de données/d'utilisation octet 2 bit 0', class Errors, trigger "WP231PR_DB_s_IO_DATA_DATA_CMD_ERROR_1" bit 8
   107: '5103 Befehl nicht möglich, da Eichanzeige fehlt oder nicht sichtbar / 5103 Command not possible - SecureDisplay is missing or hidden / 5103 Ordre impossible parce que l'afficheur légal manque ou n'est pas disponible', class Errors, trigger "WP231PR_DB_s_IO_DATA_DATA_CMD_ERROR_1" bit 9
   108: '5101 Befehle in diesem Zustand nicht möglich / 5101 Command in this state not possible / 5101 Ordre impossible dans cet état', class Errors, trigger "WP231PR_DB_s_IO_DATA_DATA_CMD_ERROR_1" bit 10
   109: '5104 Befehl nicht möglich, da Bereich überschritten / 5104 Command not possible - Limit exceeded / 5104 Ordre impossible parce que la plage de mesure est dépassée', class Errors, trigger "WP231PR_DB_s_IO_DATA_DATA_CMD_ERROR_1" bit 12
   110: 'Technologiefehlerbyte 2 Bit 7 / Technological error Byte 2 Bit 7 / Erreur technologique octet 2 bit 7', class Errors, trigger "WP231PR_DB_s_IO_DATA_TECHNOLOGICAL_ERRORS" bit 15
   111: '5105 Wägezellenparameter nicht plausibel / 5105 Load cell parameter not plausible / 5105 Les paramètres pesons ne sont pas plausibles', class Errors, trigger "WP231PR_DB_s_IO_DATA_DATA_CMD_ERROR_1" bit 13
   112: '5107 Kennlinienverschiebung nicht möglich / 5107 Calibration charcteristic shift not possible / 5107 Translation de la courbe caractéristique impossible', class Errors, trigger "WP231PR_DB_s_IO_DATA_DATA_CMD_ERROR_1" bit 15
   113: '5109 Protokollierung nicht möglich, da seit letzter Protokollierung keine Messwertänderung stattgefunden hat / 5109 Logging not possible, as the weight value did not change since the last logging / 5109 Mémorisation du rapport impossible parceque le poids n'a pas changé depuis le dernier rapport', class Errors, trigger "WP231PR_DB_s_IO_DATA_DATA_CMD_ERROR_2" bit 0
   114: 'Daten-Bedienfehler Byte 2 Bit 0 / Data Command Error Byte 3 Bit 1 / Erreur de données/d'utilisation octet 3 bit 1', class Errors, trigger "WP231PR_DB_s_IO_DATA_DATA_CMD_ERROR_2" bit 1
   115: 'Daten-Bedienfehler Byte 2 Bit 0 / Data Command Error Byte 3 Bit 2 / Erreur de données/d'utilisation octet 3 bit 2', class Errors, trigger "WP231PR_DB_s_IO_DATA_DATA_CMD_ERROR_2" bit 2
   116: 'Daten-Bedienfehler Byte 2 Bit 0 / Data Command Error Byte 3 Bit 3 / Erreur de données/d'utilisation octet 3 bit 3', class Errors, trigger "WP231PR_DB_s_IO_DATA_DATA_CMD_ERROR_2" bit 3
   117: 'Daten-Bedienfehler Byte 2 Bit 0 / Data Command Error Byte 3 Bit 4 / Erreur de données/d'utilisation octet 3 bit 4', class Errors, trigger "WP231PR_DB_s_IO_DATA_DATA_CMD_ERROR_2" bit 4
   118: '5199 Fehler bei Befehl an DE / 5199 Error caused by command on DI / 5199 Erreur d'ordre entré par une entrée TOR', class Errors, trigger "WP231PR_DB_s_IO_DATA_DATA_CMD_ERROR_2" bit 5
   119: 'Daten-Bedienfehler Byte 2 Bit 0 / Erreur de données/d'utilisation octet 3 bit 6', class Errors, trigger "WP231PR_DB_s_IO_DATA_DATA_CMD_ERROR_2" bit 6
   120: 'Daten-Bedienfehler Byte 2 Bit 0 / Data Command Error Byte 3 Bit 7 / Erreur de données/d'utilisation octet 3 bit 7', class Errors, trigger "WP231PR_DB_s_IO_DATA_DATA_CMD_ERROR_2" bit 7
   121: 'Daten-Bedienfehler Byte 4 Bit 0 / Data Command Error Byte 4 Bit 0 / Erreur de données/d'utilisation octet 4 bit 0', class Errors, trigger "WP231PR_DB_s_IO_DATA_DATA_CMD_ERROR_2" bit 8
   122: 'Daten-Bedienfehler Byte 4 Bit 1 / Data Command Error Byte 4 Bit 1 / Erreur de données/d'utilisation octet 4 bit 1', class Errors, trigger "WP231PR_DB_s_IO_DATA_DATA_CMD_ERROR_2" bit 9
   123: 'Daten-Bedienfehler Byte 4 Bit 2 / Data Command Error Byte 4 Bit 2 / Erreur de données/d'utilisation octet 4 bit 2', class Errors, trigger "WP231PR_DB_s_IO_DATA_DATA_CMD_ERROR_2" bit 10
   124: 'Daten-Bedienfehler Byte 2 Bit 0 / Data Command Error Byte 2 Bit 6 / Erreur de données/d'utilisation octet 2 bit 6', class Errors, trigger "WP231PR_DB_s_IO_DATA_DATA_CMD_ERROR_1" bit 14
   125: 'Technologiefehlerbyte 2 Bit 6 / Technological error Byte 2 Bit 6 / Erreur technologique octet 2 bit 6', class Errors, trigger "WP231PR_DB_s_IO_DATA_TECHNOLOGICAL_ERRORS" bit 14
   126: 'Technologiefehlerbyte 2 Bit 5 / Technological error Byte 2 Bit 5 / Erreur technologique octet 2 bit 5', class Errors, trigger "WP231PR_DB_s_IO_DATA_TECHNOLOGICAL_ERRORS" bit 13
   127: 'Technologiefehlerbyte 2 Bit 4 / Technological error Byte 2 Bit 4 / Erreur technologique octet 2 bit 4', class Errors, trigger "WP231PR_DB_s_IO_DATA_TECHNOLOGICAL_ERRORS" bit 12
   128: '1000 Betriebsfehler liegt vor / 1000 Operation Error / 1000 Erreur de fonctionnement', class Errors, trigger "WP231PR_DB_s_IO_DATA_OPERATION_ERRORS" bit 0
   129: 'Betriebsfehler Byte 1 Bit 1 / Operation Error Byte 1 Bit 1 / 1101 Court circuit pesons', class Errors, trigger "WP231PR_DB_s_IO_DATA_OPERATION_ERRORS" bit 1
   130: '1104 ADC Sense-Spannung zu gering / 1104 ADC sense voltage too low / 1104 Tension capteurs CAN trop basse', class Errors, trigger "WP231PR_DB_s_IO_DATA_OPERATION_ERRORS" bit 2
   131: 'Betriebsfehler Byte 1 Bit 3 / Operation Error Byte 1 Bit 1 / 1101 Court circuit pesons', class Errors, trigger "WP231PR_DB_s_IO_DATA_OPERATION_ERRORS" bit 3
   5: '1105 ADC Ausserhalb zulässigem Digit-Bereich (positiv) / 1105 ADC out of range (positive) / 1105 CAN hors plage de mesure (max)', class Errors, trigger "WP231PR_DB_s_IO_DATA_OPERATION_ERRORS" bit 4
   6: '1106 ADC Ausserhalb zulässigem Digit-Bereich (negativ) / 1106 ADC out of range (negative) / 1106 CAN hors plage de mesure (min)', class Errors, trigger "WP231PR_DB_s_IO_DATA_OPERATION_ERRORS" bit 5
   132: '1002 RAM-Fehler / 1002 RAM error / 1002 Erreur RAM', class Errors, trigger "WP231PR_DB_s_IO_DATA_OPERATION_ERRORS" bit 6
   133: '1102 ADC Fehler / 1102 ADC error / 1102 Erreur CAN', class Errors, trigger "WP231PR_DB_s_IO_DATA_OPERATION_ERRORS" bit 7
   134: '1005 Prozessalarm verloren / 1005 Processalarm lost / 1005 Perte des messages processus', class Errors, trigger "WP231PR_DB_s_IO_DATA_OPERATION_ERRORS" bit 8
   135: '1003 Checksummenfehler Daten / 1003 Checksum error data / 1003 Erreur données checksum', class Errors, trigger "WP231PR_DB_s_IO_DATA_OPERATION_ERRORS" bit 9
   136: '1107 Eichfähige HMI-Anzeige ist ausgefallen / 1107 Legal-for-trade display disturbed / 1107 Perte de l'affichage légal sur le pupitre HMI', class Errors, trigger "WP231PR_DB_s_IO_DATA_OPERATION_ERRORS" bit 10
   137: '1004 Checksummenfehler Programm / 1004 Checksum error program / 1004 Erreur données checksum du programme', class Errors, trigger "WP231PR_DB_s_IO_DATA_OPERATION_ERRORS" bit 11
   138: '1001 Reset nach Fehler (Watchdog Error) / 1001 Restart after failure (watchdog error) / 1001 Reset après erreur (Watchdog)', class Errors, trigger "WP231PR_DB_s_IO_DATA_OPERATION_ERRORS" bit 13
   139: '1007 Falsche Applikations-ID / 1007 Wrong application ID / 1007 Erreur ID de l'application', class Errors, trigger "WP231PR_DB_s_IO_DATA_OPERATION_ERRORS" bit 14
   140: 'Betriebsfehlerbyte 2 Bit 7 / Operation Error Byte 2 Bit 7 / Erreur fonctionnement octet 2 bit 7', class Errors, trigger "WP231PR_DB_s_IO_DATA_OPERATION_ERRORS" bit 15
   141: '2000 Technologiefehler / 2000 Technological error / 2000 Erreur technologique', class Errors, trigger "WP231PR_DB_s_IO_DATA_TECHNOLOGICAL_ERRORS" bit 0
   142: '2001 Timeout Tarieren oder Nullstellen / 2001 Timeout tare or zero setting / 2001 Timeout tarage ou RAZ (temps d'attente dépassé)', class Errors, trigger "WP231PR_DB_s_IO_DATA_TECHNOLOGICAL_ERRORS" bit 1
   143: '2002 Trace überlastet / 2002 Trace overloaded / 2002 Mémoire trace pleine', class Errors, trigger "WP231PR_DB_s_IO_DATA_TECHNOLOGICAL_ERRORS" bit 2
   144: '2003 Einschaltnullsetzen nicht möglich / 2003 Initial Zeroing not possible / 2003 RAZ à la mise sous tension impossible', class Errors, trigger "WP231PR_DB_s_IO_DATA_TECHNOLOGICAL_ERRORS" bit 3
   145: 'Technologiefehlerbyte 1 Bit 4 / Technological error Byte 1 Bit 4 / Erreur technologique octet 1 bit 4', class Errors, trigger "WP231PR_DB_s_IO_DATA_TECHNOLOGICAL_ERRORS" bit 4
   146: 'Technologiefehlerbyte 1 Bit 5 / Technological error Byte 1 Bit 5 / Erreur technologique octet 1 bit 5', class Errors, trigger "WP231PR_DB_s_IO_DATA_TECHNOLOGICAL_ERRORS" bit 5
   147: 'Technologiefehlerbyte 1 Bit 6 / Technological error Byte 1 Bit 6 / Erreur technologique octet 1 bit 6', class Errors, trigger "WP231PR_DB_s_IO_DATA_TECHNOLOGICAL_ERRORS" bit 6
   148: 'Technologiefehlerbyte 1 Bit 7 / Technological error Byte 1 Bit 7 / Erreur technologique octet 1 bit 7', class Errors, trigger "WP231PR_DB_s_IO_DATA_TECHNOLOGICAL_ERRORS" bit 7
   149: 'Technologiefehlerbyte 1 Bit 7 / Technological error Byte 2 Bit 0 / Erreur technologique octet 2 bit 0', class Errors, trigger "WP231PR_DB_s_IO_DATA_TECHNOLOGICAL_ERRORS" bit 8
   150: 'Technologiefehlerbyte 2 Bit 1 / Technological error Byte 2 Bit 1 / Erreur technologique octet 2 bit 1', class Errors, trigger "WP231PR_DB_s_IO_DATA_TECHNOLOGICAL_ERRORS" bit 9
   151: 'Technologiefehlerbyte 2 Bit 2 / Technological error Byte 2 Bit 2 / Erreur technologique octet 2 bit 2', class Errors, trigger "WP231PR_DB_s_IO_DATA_TECHNOLOGICAL_ERRORS" bit 10
   152: 'Technologiefehlerbyte 2 Bit 3 / Technological error Byte 2 Bit 3 / Erreur technologique octet 2 bit 3', class Errors, trigger "WP231PR_DB_s_IO_DATA_TECHNOLOGICAL_ERRORS" bit 11
   153: '6002 Protokollieren nicht möglich, da Gewicht unzulässig / 6002 Logging not possible - Weight not plausible / 6002 Impossible d'écrire le rapport, le poids est hors tolérances', class Errors, trigger "WP231PR_DB_s_IO_DATA_DATA_CMD_ERROR_2" bit 11
   61: '5108 Logbuch-ID nicht vorhanden / 5108 Log ID not existing / 5108 Carnet de rapport n'existe pas', class Errors, trigger "WP231PR_DB_s_IO_DATA_DATA_CMD_ERROR_2" bit 12
   154: '5102 Befehl nicht möglich, da kein Stillstand vorliegt / 5102 Command not possible - No Standstill / 5102 Ordre impossible parce que l'état stable n'est pas atteint', class Errors, trigger "WP231PR_DB_s_IO_DATA_DATA_CMD_ERROR_1" bit 11
   63: 'Daten-Bedienfehler Byte 4 Bit 2 / Data Command Error Byte 4 Bit 6 / Erreur de données/d'utilisation octet 4 bit 6', class Errors, trigger "WP231PR_DB_s_IO_DATA_DATA_CMD_ERROR_2" bit 14
   81: '7017 MAC Adresse kann nicht geändert werden / 7017 MAC address can not be changed / 7017 Impossible de changer l'adresse MAC', class Errors, trigger "WP231PR_DB_s_IO_DATA_DATA_CMD_ERROR_4" bit 0
   82: '7018 Fehler in IP-Maske / 7018 Error in IP mask / 7018 Erreur dans la vue IP', class Errors, trigger "WP231PR_DB_s_IO_DATA_DATA_CMD_ERROR_4" bit 1
   83: '7019 RS485 Parameter nicht plausibel / 7019 RS485 parameter not plausible / 7019 Les paramètres RS485 ne sont pas plausibles', class Errors, trigger "WP231PR_DB_s_IO_DATA_DATA_CMD_ERROR_4" bit 2
   84: 'Daten-Bedienfehler Byte 7 Bit 4 / Data- / Command Error Byte 7 Bit 3 / Erreur de données/d'utilisation octet 7 bit 3', class Errors, trigger "WP231PR_DB_s_IO_DATA_DATA_CMD_ERROR_4" bit 3
   85: 'Daten-Bedienfehler Byte 7 Bit 5 / Data- / Command Error Byte 7 Bit 4 / Erreur de données/d'utilisation octet 7 bit 4', class Errors, trigger "WP231PR_DB_s_IO_DATA_DATA_CMD_ERROR_4" bit 4
   86: 'Daten-Bedienfehler Byte 7 Bit 6 / Data- / Command Error Byte 7 Bit 5 / Erreur de données/d'utilisation octet 7 bit 5', class Errors, trigger "WP231PR_DB_s_IO_DATA_DATA_CMD_ERROR_4" bit 5
   87: 'Daten-Bedienfehler Byte 7 Bit 7 / Data- / Command Error Byte 7 Bit 6 / Erreur de données/d'utilisation octet 7 bit 6', class Errors, trigger "WP231PR_DB_s_IO_DATA_DATA_CMD_ERROR_4" bit 6
   80: '7016 Parametrierung des Analogausgangs ist nicht plausibel / 7016 Analog output parameter not plausible / 7016 Le paramétrage de la sortie analogique n'est pas plausible', class Errors, trigger "WP231PR_DB_s_IO_DATA_DATA_CMD_ERROR_3" bit 15
   88: 'Daten-Bedienfehler Byte 8 Bit 0 / Data- / Command Error Byte 7 Bit 7 / Erreur de données/d'utilisation octet 7 bit 7', class Errors, trigger "WP231PR_DB_s_IO_DATA_DATA_CMD_ERROR_4" bit 7
   91: 'Daten-Bedienfehler Byte 8 Bit 3 / Data- / Command Error Byte 8 Bit 2 / Erreur de données/d'utilisation octet 8 bit 2', class Errors, trigger "WP231PR_DB_s_IO_DATA_DATA_CMD_ERROR_4" bit 10
   92: 'Daten-Bedienfehler Byte 8 Bit 4 / Data- / Command Error Byte 8 Bit 3 / Erreur de données/d'utilisation octet 8 bit 3', class Errors, trigger "WP231PR_DB_s_IO_DATA_DATA_CMD_ERROR_4" bit 11
   93: 'Daten-Bedienfehler Byte 8 Bit 5 / Data- / Command Error Byte 8 Bit 4 / Erreur de données/d'utilisation octet 8 bit 4', class Errors, trigger "WP231PR_DB_s_IO_DATA_DATA_CMD_ERROR_4" bit 12
   94: 'Daten-Bedienfehler Byte 8 Bit 6 / Data- / Command Error Byte 8 Bit 5 / Erreur de données/d'utilisation octet 8 bit 5', class Errors, trigger "WP231PR_DB_s_IO_DATA_DATA_CMD_ERROR_4" bit 13
   95: 'Daten-Bedienfehler Byte 8 Bit 6 / Data- / Command Error Byte 8 Bit 6 / Erreur de données/d'utilisation octet 8 bit 6', class Errors, trigger "WP231PR_DB_s_IO_DATA_DATA_CMD_ERROR_4" bit 14
   96: 'Daten-Bedienfehler Byte 8 Bit 6 / Data- / Command Error Byte 8 Bit 6 / Erreur de données/d'utilisation octet 8 bit 7', class Errors, trigger "WP231PR_DB_s_IO_DATA_DATA_CMD_ERROR_4" bit 15
   62: 'Daten-Bedienfehler Byte 4 Bit 2 / Data Command Error Byte 4 Bit 5 / Erreur de données/d'utilisation octet 4 bit 5', class Errors, trigger "WP231PR_DB_s_IO_DATA_DATA_CMD_ERROR_2" bit 13
   89: 'Daten-Bedienfehler Byte 8 Bit 1 / Data- / Command Error Byte 8 Bit 0 / Erreur de données/d'utilisation octet 8 bit 0', class Errors, trigger "WP231PR_DB_s_IO_DATA_DATA_CMD_ERROR_4" bit 8
   79: 'Daten-Bedienfehler Byte 6 Bit 6 / Data- / Command Error Byte 6 Bit 6 / Erreur de données/d'utilisation octet 6 bit 6', class Errors, trigger "WP231PR_DB_s_IO_DATA_DATA_CMD_ERROR_3" bit 14
   90: 'Daten-Bedienfehler Byte 8 Bit 2 / Data- / Command Error Byte 8 Bit 1 / Erreur de données/d'utilisation octet 8 bit 1', class Errors, trigger "WP231PR_DB_s_IO_DATA_DATA_CMD_ERROR_4" bit 9
   78: '7014 Zeitvorgabe nicht plausibel / 7014 Time value not plausible / 7014 de données/d'utilisation octet 6 bit 5', class Errors, trigger "WP231PR_DB_s_IO_DATA_DATA_CMD_ERROR_3" bit 13
   65: '7000 Zulässiger Zahlenbereich verlassen / 7000 Counting range exceeded / 7000 Hors plage numérique', class Errors, trigger "WP231PR_DB_s_IO_DATA_DATA_CMD_ERROR_3" bit 0
   66: 'Daten-Bedienfehler Byte 5 Bit 1 / Data Command Error Byte 5 Bit 1 / Erreur de données/d'utilisation octet 5 bit 1', class Errors, trigger "WP231PR_DB_s_IO_DATA_DATA_CMD_ERROR_3" bit 1
   67: '7001 Vorschriftencode nicht bekannt / 7001 Restriction code unknown / 7001 Code métrologique inconnu', class Errors, trigger "WP231PR_DB_s_IO_DATA_DATA_CMD_ERROR_3" bit 2
   69: '7003 Vorgabe Datum/Uhrzeit nicht plausibel / 7003 Date / Time parameter not plausible / 7003 Consigne de date/heure pas plausible', class Errors, trigger "WP231PR_DB_s_IO_DATA_DATA_CMD_ERROR_3" bit 4
   70: '7004 Zuordnung DQ/DI nicht plausibel / 7004 Assignment of digital input or output not plausible / 7004 Affectation des entrées/sorties TOR erronée', class Errors, trigger "WP231PR_DB_s_IO_DATA_DATA_CMD_ERROR_3" bit 5
   71: 'Daten-Bedienfehler Byte 5 Bit 6 / Data- / Command Error Byte 5 Bit 6 / 7006 Ordre réservé pour banc de test usine', class Errors, trigger "WP231PR_DB_s_IO_DATA_DATA_CMD_ERROR_3" bit 6
   72: '7007 Die Justagegewichte bzw. Justagedigits sind nicht plausibel / 7007 Calibrationweights / Calibrationdigits not plausible / 7007 Les poids étalons ou les digits d'étalonnage ne sont pas plausibles', class Errors, trigger "WP231PR_DB_s_IO_DATA_DATA_CMD_ERROR_3" bit 7
   68: 'Daten-Bedienfehler Byte 5 Bit 3 / Data Command Error Byte 5 Bit 3 / Erreur de données/d'utilisation octet 5 bit 1', class Errors, trigger "WP231PR_DB_s_IO_DATA_DATA_CMD_ERROR_3" bit 3
   74: '7009 Stillstandsbereich / Stillstandswartezeit nicht plausibel / 7009 Standstillrange / Standstilltime not plausible / 7009 Les valeurs de tempo ou de poids pour l'état stable ne sont pas plausibles', class Errors, trigger "WP231PR_DB_s_IO_DATA_DATA_CMD_ERROR_3" bit 9
   73: '7008 Nullstell- / Nullsetz- oder Taraparameter nicht plausibel / 7008 Zero- / Tare weights not plausible / 7008 Les valeur de RAZ ne sont pas plausibles', class Errors, trigger "WP231PR_DB_s_IO_DATA_DATA_CMD_ERROR_3" bit 8
   77: '7013 Schnittstellenparameter SecureDisplay nicht plausibel / 7013 Interface settings for legal display not plausible / 7013 Les paramètres de SecureDisplay ne sont pas plausibles', class Errors, trigger "WP231PR_DB_s_IO_DATA_DATA_CMD_ERROR_3" bit 12
   76: '7011 Filterparameter nicht plausibel / 7011 Filter parameter not plausible / 7011 Les paramètres des filtres ne sont pas plausibles', class Errors, trigger "WP231PR_DB_s_IO_DATA_DATA_CMD_ERROR_3" bit 11
   64: 'Daten-Bedienfehler Byte 4 Bit 2 / Data Command Error Byte 4 Bit 7 / Erreur de données/d'utilisation octet 4 bit 7', class Errors, trigger "WP231PR_DB_s_IO_DATA_DATA_CMD_ERROR_2" bit 15
   75: '7010 Ziffernschritt / Rundung nicht plausibel / 7010 Numeral step / rounding not plausible / 7010 Echelon ou arrondit ne sont pas plausibles', class Errors, trigger "WP231PR_DB_s_IO_DATA_DATA_CMD_ERROR_3" bit 10

text list "Hand": 0 'Авто'; 1 'Ручной'

text list "003030_LETTER_FOR_GROSS_WEIGHT": 66 'B für Brutto / B for Gross / B pour Brut'; 71 'G für Brutto / G for Gross / G pour Brut'

graphic list "ok": 0 'check_box_off'; 1 'check_box_on'

graphic list "Motor": 0 'm_off_1'; 1 'm_on_1'; 2..8 'm_wait_1'; 9..1000 'm_alarm_1'

graphic list "ON_OFF": 0 'off_toggle'; 1 'on_toggle'

graphic list "Alarm": 0 'no_alarm_1'; 1 'alarm'

graphic list "Valve": 0 'v_off'; 1 'v_on'; 2..8 'v_wait'; 9..1000 'v_alarm'

graphic list "Signal_grey_yellow": 1 'Field Yellow'; 0 'Field Grey'

